(* CODESYS project shutter.library
   Company: ESO
   Description: Local Device Control - LDC Shutter Library based on State Machine
   Version: 1.1.1.0
   Placeholder: ESO LDC Shutter Library
   Author: Dan Popovic
   Title: ESO LDC Shutter Library

Project tree, tasks and I/O mapping:
  libraries: Tc2_Standard, * (Beckhoff Automation GmbH); Tc2_System, * (Beckhoff Automation GmbH); Tc3_EventLogger, * (Beckhoff Automation GmbH); Tc3_Module, * (Beckhoff Automation GmbH); VisuDialogs, * (System); VisuSymbols, 3.5.10.0 (System)
  config/
    Device1_EtherCAT_SPLC014.xti
    Mappings_HW_SPLC014.xml
    Mappings_SIM.xml
  00000000-0000-0000-0000-000000000000|config\Device1_EtherCAT_SPLC014.xti
  00000000-0000-0000-0000-000000000000|config\Mappings_HW_SPLC014.xml
  00000000-0000-0000-0000-000000000000|config\Mappings_SIM.xml
  doc/
  DUTs/
    Enumerated/
      data type E_SHUTTER_COMMAND
      data type E_SHUTTER_ERROR
      data type E_SHUTTER_EVENT
      data type E_SHUTTER_HW_STATUS
      data type E_SHUTTER_RPC_ERROR
      data type E_SHUTTER_STATE
      data type E_SHUTTER_STATUS
      data type E_SHUTTER_SUBSTATE
    Structures/
      data type T_SHUTTER_CFG
      data type T_SHUTTER_CTRL
      data type T_SHUTTER_INFO
      data type T_SHUTTER_STAT
      data type T_SIM_SHUTTER_CFG
      data type T_SIM_SHUTTER_STAT
  GVLs/
  lib/
  POUs/
    function block FB_SHUTTER [ST]: ActionCloseExecute, ActionDisableComplete, ActionDisableExecute, ActionEnableComplete, ActionErrExecute, ActionInitAbort, ActionInitComplete, ActionInitExecute, ActionInitReject, ActionOpenExecute, ActionResetExecute, ActionStopExecute, ActionUnexpExecute, ActivityClosing, ActivityDisabling, ActivityInitializing, ActivityOpening, CheckForEvents, M_GetLogicalState, M_GetRpcErrorText, M_SetLastCommand, M_SetRpcStatus, RPC_Close, RPC_Disable, RPC_Enable, RPC_Init, RPC_Open, RPC_Reset, RPC_SetDebug, RPC_SetLog, RPC_Stop
    function block FB_SHUTTER_BASE [ST]: ActionCloseExecute, ActionDisableExecute, ActionEnableComplete, ActionEnableExecute, ActionErrExecute, ActionInitAbort, ActionInitComplete, ActionInitExecute, ActionInitReject, ActionOpenExecute, ActionResetExecute, ActionStopExecute, ActionUnexpExecute, ActivityClosing, ActivityDisabling, ActivityInitializing, ActivityOpening, CheckForEvents, M_Configure, M_GetErrorText, M_LogEventDebug, M_LogEventEnd, M_LogEventError, M_LogEventGeneral, M_LogEventStart, M_SetStatus, ProcessEvents, SetAction, SetEvent, SetState
    function block FB_SIM_SHUTTER [ST]: M_GetLogicalState, RPC_ResetConfig, RPC_SetActiveLow_Closed, RPC_SetActiveLow_Fault, RPC_SetActiveLow_Open, RPC_SetActiveLow_Switch, RPC_SetCouplerState, RPC_SetDelay, RPC_SetFault, SetState
    program MAIN [ST]
  Version/
    global variables Global_Version
  VISUs/
    Templates/
      visualisation GUI_TEMPLATE_SHUTTER
    visualisation GUI_All
    visualisation GUI_Shutter001
  text list GlobalTextList
  00000000-0000-0000-0000-000000000000|Shutter.tmc
  Shutter.tmc
*)

// DUTs/Enumerated/E_SHUTTER_COMMAND
{attribute 'qualified_only'}
{attribute 'strict'}
TYPE E_SHUTTER_COMMAND :
(
	NONE	:= 0,
	
	RESET,
	INIT,
	STOP,
	ENABLE,
	DISABLE,
	OPEN,
	CLOSE
	
);
END_TYPE

// DUTs/Enumerated/E_SHUTTER_ERROR
{attribute 'qualified_only'}
{attribute 'strict'}
TYPE E_SHUTTER_ERROR :
(
	OK						:= 0,
	HW_NOT_OP,			
	INIT_FAILURE,		
	UNEXPECTED_CLOSED,
	UNEXPECTED_NONE,
	UNEXPECTED_OPENED,
	FAULT_SIG,
	BOTH_SIG_ACTIVE,
	TIMEOUT_ENABLE,
	TIMEOUT_DISABLE,
	TIMEOUT_INIT,
	TIMEOUT_CLOSE,
	TIMEOUT_OPEN,

	SIM_NOT_INITIALISED		:= 90,
	SIM_NULL_POINTER			:= 100	// Simulator error
);
END_TYPE

// DUTs/Enumerated/E_SHUTTER_EVENT
{attribute 'qualified_only'}
{attribute 'strict'}
TYPE E_SHUTTER_EVENT :
(
	NONE	:= 0,
	
	(* events corresponding to commands *)
	RESET,
	INIT,
	STOP,
	ENABLE,
	DISABLE,
	OPEN,
	CLOSE,
	
	(* 
		Events corresponding to internal events 
	*)
	
	INITOPEN,		// Needed for detection of HW failures during initialisation
	INITCLOSED,
	DISABLEOPEN,
	DISABLECLOSED,
	
	(* events mapped to HW signals *)
	ISOPEN,
	ISCLOSED,

	HWOK,
	ERRHW,
	ERRFAULT,
	ERRALLACTIVE,
	ERRNONEACTIVE,	
	ERRINIT,
	ERRDISABLE,
	ERRTIMEOUTCLOSE,
	ERRTIMEOUTOPEN
	
);
END_TYPE

// DUTs/Enumerated/E_SHUTTER_HW_STATUS
{attribute 'qualified_only'}
{attribute 'strict'}
TYPE E_SHUTTER_HW_STATUS :
(
	UNKNOWN	:= 0,
	ERROR,
	CLOSED,
	OPEN
);
END_TYPE

// DUTs/Enumerated/E_SHUTTER_RPC_ERROR
{attribute 'qualified_only'}
{attribute 'strict'}
TYPE E_SHUTTER_RPC_ERROR :
(
	OK					:= 0,
	NOT_OP				:= -1,			
	NOT_NOTOP_READY		:= -2,			
	NOT_NOTOP_NOTREADY	:= -3,			
	STILL_OPENING		:= -4,			
	STILL_CLOSING		:= -5,			
	LOCAL				:= -6			
);
END_TYPE

// DUTs/Enumerated/E_SHUTTER_STATE
{attribute 'qualified_only'}
{attribute 'strict'}
TYPE E_SHUTTER_STATE :
(
	NONE	:= 0,
	NOTOP,
	OP
);
END_TYPE

// DUTs/Enumerated/E_SHUTTER_STATUS
{attribute 'qualified_only'}
{attribute 'strict'}
TYPE E_SHUTTER_STATUS :
(
	OK	:= 0,
	ERROR
);
END_TYPE

// DUTs/Enumerated/E_SHUTTER_SUBSTATE
{attribute 'qualified_only'}
{attribute 'strict'}
TYPE E_SHUTTER_SUBSTATE :
(
	NONE                 	:= 0,
	
	NOTOP_NOTREADY     		:= 100,
	NOTOP_INITIALIZING		:= 102,
	NOTOP_READY_CLOSED		:= 105,
	NOTOP_READY_OPEN		:= 106,
	NOTOP_ERROR				:= 199,
	
	OP_DISABLING         	:= 205,
	OP_CLOSED				:= 212,            
	OP_CLOSING				:= 213,           
	OP_OPEN					:= 214,
	OP_OPENING				:= 215,
	OP_ERROR				:= 299
);
END_TYPE

// DUTs/Structures/T_SHUTTER_CFG
TYPE T_SHUTTER_CFG :
STRUCT
	sName:				STRING	:= 'Shutter';	// Instance name

	bActiveLowClosed:	BOOL 	:= FALSE;		// If TRUE, the CLOSED signal is Active Low, default FALSE
	bActiveLowFault:	BOOL 	:= FALSE;		// If TRUE, the FAULT signal is Active Low, default FALSE
	bActiveLowOpen:		BOOL 	:= FALSE;		// If TRUE, the OPEN signal is Active Low, default FALSE
	bActiveLowSwitch:	BOOL 	:= FALSE;		// If TRUE, the SWITCH signal is Active Low, default FALSE

	bIgnoreClosed:		BOOL 	:= FALSE;		// If TRUE, the CLOSED signal is Ignored, default FALSE
	bIgnoreFault:		BOOL 	:= FALSE;		// If TRUE, the FAULT signal is Ignored, default FALSE
	bIgnoreOpen:		BOOL 	:= FALSE;		// If TRUE, the OPEN signal is Ignored, default FALSE

	bInitialState:		BOOL 	:= FALSE;		// Default shutter position is FALSE/CLOSED
	nTimeout:     		UDINT 	:= 3000;		// Timeout for OPEN/CLOSE transitions [msec], default 3000 ms
	
	// Logging
	bLogExtTime:		BOOL 	:= FALSE;		// If TRUE, use external time in event logs. Default FALSE.
	bDebug:				BOOL 	:= FALSE;		// If TRUE, show event logs of Debug type. Default FALSE.
	bLog:				BOOL 	:= TRUE;		// If TRUE, log events. Default TRUE.
	
END_STRUCT
END_TYPE

// DUTs/Structures/T_SHUTTER_CTRL
TYPE T_SHUTTER_CTRL :
STRUCT
	nCommand:	E_SHUTTER_COMMAND	:= E_SHUTTER_COMMAND.NONE; (* See E_SHUTTER_COMMAND *)
	bExecute:	BOOL;
	
END_STRUCT
END_TYPE

// DUTs/Structures/T_SHUTTER_INFO
TYPE T_SHUTTER_INFO :
STRUCT
(*
Driver Information 

Change Log:
	0.1	2015-12-11	- First version - dummy implementation.
	0.2	2015-12-15	- Added timer for dummy initialization. Cleanup.
	0.3	2015-12-15	- One method per state.
	0.4	2016-06-24	- Transfer of code from FB_SHUTTER (VLT code).
	0.6 2016-06-30	- OPC UA Read Only for info and stat.
					- New method: GetLogicalState() to replace F_GET_LOGICAL_STATE
					  coming from TC3 Common.library.
					- Removed Common.library from References.
					- Implemented simulator FB_SIM_SHUTTER.
					- References are 'Always Newest'.
					- Removed Recording project.
	0.7 2016-07-01	- Added RPC_SetCouplerState() in FB_SIM_SHUTTER.
					- OPC UA Configuration cleanup
					- Removed FB_SHUTTER_SIM.
	0.8 2016-07-01	- Renaming from *_SHUTTER_* to *_SHUTTER_*.
					- Restructuring of GUI.
					- Addition of GUI Template.
					- Addition of sName as FB_SHUTTER input parameter.
					- Addition of Shutter.library
	0.9 2016-07-12	- Addition of method ActionResetExecute().
					- Errors updated only if it is currently equal to OK.
	0.10 2016-07-13	- bOpen and bClosed determined taking into account configuration.
	0.11 2017-01-25	- Addition of stat.sLastCommand.
					- Adopted Simulator from VLT FB_SIM_SHUTTER.
	0.12 2017-08-07	- Addition of BOOL return value for all RPC Calls.
					- Addition of stat.sRPCErrorText variable.
	0.13 2017-08-25	- Improved RPC Calls for all possible failures.
	0.14 2017-08-25	- Removed E_SHUTTER_SUBSTATE.NOTOP_READY substate.
					- Fixed RPC_Enable bug.
	0.15.0.0		- Single pointer to simulator
					- Updated Visualisation version
	0.16.0.0		- Corrected Simulator handling of Update.
					- Removed bUpdate variable from Simulator.
					- Addition of SetState() Simulator method.
	0.17.0.0		- Simulator delay set to half real shutter timeout.
	0.18.0.0		- Addition of all cfg params as input params.
					- Addition of M_Configure() in FB_SHUTTER_BASE.
					- Added return value for Simulator RPC calls.
					- Added small delay to simulator on re-boot.
					- Moved sName to cfg structure.
					- Single GUI for all shutters.
	0.19.0.0		- Addition of measured times for open/close in T_SHUTTER_STAT.
	0.20.0.0		- Addition of stat.sLibVersion
	0.21.0.0		- RPC calls return INT.
					- Addition of E_SHUTTER_RPC_ERROR.
	0.22.0.0		- Addition of M_GetRpcErrorText().
					- Addition of M_SetRpcStatus().
					- Improved template GUI.
					- Addition of M_GetErrorText().
					- M_SetStatus() replaced SetStatus().
					- Improved error handling.
	0.22.0.1		- Addition of library category ESO/ELT.
	0.23.0.0		- Renaming States STANDBY->NOTOP & FAILURE->ERROR.
					- RPC commands rejected in Local mode.
	0.23.0.1		- Corrected handling of IgnoreFault.
	1.0.0.0			- WARNING: Requires TwinCAT 3.1 build 4022.20 or higher.
					- Projects need Tc3_EventLogger library included in References.
					- Addition of Methods for Event Logs.
					- Addition of method RPC_Debug().
	1.0.0.1			- Addition of cfg.bLog flag for enable/disable of logging.
					- Renamed RPC_Debug() to RPC_SetDebug().
					- Addition of RPC_SetLog().
	1.0.0.2			- Compiled wit TwinCAT 3.1 build 4022.27.
					- Renamed TC_EVENTS.OpsEventClass to TC_EVENTS.ShutterOpsEventClass.
					- Solved problem of 'growing' libraries by setting Property/Advanced/BuildAction to None for Shutter.library.
					- Pinned ST_ShutterOpsEventClass under External Types.
	1.1.0.0			- Using Strict enumerations.
*)
	sDate:			STRING(32)	:= '2019-04-25';
	sDescription:	STRING(80) 	:= 'State Machine based Shutter controller';
	sName:			STRING(64)	:= 'FB_SHUTTER';
	sPlatform:		STRING(32)	:= 'CoDeSys';
	sSynopsis:		STRING(64)	:= 'State Machine based Shutter controller';
	nVersionMajor:	DINT		:= 1;
	nVersionMinor:	DINT		:= 1;
END_STRUCT
END_TYPE

// DUTs/Structures/T_SHUTTER_STAT
TYPE T_SHUTTER_STAT :
STRUCT
	//
	// Common variables START
	//
	bLocal:			BOOL	:= FALSE;						(* Device operated from PLC GUI *)

	nState:			E_SHUTTER_STATE		:= E_SHUTTER_STATE.NOTOP;			(* State, see E_SHUTTER_STATE *)
	nSubstate:		E_SHUTTER_SUBSTATE	:= E_SHUTTER_SUBSTATE.NOTOP_NOTREADY;(* Substate, see E_SHUTTER_SUBSTATE *)

	nErrorCode: 	E_SHUTTER_ERROR 	:= E_SHUTTER_ERROR.OK;				(* Error code *)
	nLastCommand:	E_SHUTTER_COMMAND	:= E_SHUTTER_COMMAND.NONE;			(* Last command sent to the device *)
	nStatus: 		E_SHUTTER_STATUS	:= E_SHUTTER_STATUS.OK; 			(* Device status *)
	nHwStatus: 		E_SHUTTER_HW_STATUS	:= E_SHUTTER_HW_STATUS.UNKNOWN; 	(* Unknown, error, open, closed. See E_SHUTTER_HW_STATUS *)
	nRpcErrorCode: 	E_SHUTTER_RPC_ERROR := E_SHUTTER_RPC_ERROR.OK;			(* RPC Error code *)

	sState:			STRING	:= 'NOT OP';					(* State textual description *)
	sSubstate:		STRING	:= 'NOT READY';					(* Substate textual description *)
	sErrorText: 	STRING 	:= 'OK'; 						(* Error text *)
	sRPCErrorText: 	STRING 	:= 'OK'; 						(* RPC Error text *)
	sStatus: 		STRING 	:= 'OK'; 						(* Status in textual form, e.g. 'OFF' *)
	sHwStatus: 		STRING 	:= 'UNKNOWN'; 					(* HW Status in textual form: 'UNKNOWN', 'ERROR', 'OPEN' or 'CLOSED' *)
	sLastCommand:	STRING	:= 'NONE';						(* Last command, as string, sent to the device *)
	sLibVersion:	STRING	:= 'UNKNOWN';					(* Library version as string, e.g. '1.2.0.0' *)
	
	sActionDesc:	STRING	:= '';
	sEventDesc:		STRING	:= '';

	nCycleCounter:	UDINT	:= 0;							// Alive flag
	nCycleTime:		UDINT	:= 0;							// Cycle time in us (microsec)
	//
	// Common variables END
	//

	//
	// Device specific variables
	//
	nLastTimeToOpen:	DINT	:= -1;	// Time taken for last OPEN command [msec] (-1 = failure)
	nLastTimeToClose:	DINT	:= -1;	// Time taken for last CLOSE command [msec] (-1 = failure)
END_STRUCT
END_TYPE

// DUTs/Structures/T_SIM_SHUTTER_CFG
TYPE T_SIM_SHUTTER_CFG :
STRUCT
	bActiveLowClosed:	BOOL := FALSE;
	bActiveLowFault:	BOOL := FALSE;
	bActiveLowOpen:		BOOL := FALSE;
	bActiveLowSwitch:	BOOL := FALSE;

	nDelay:     		UDINT := 2000;	(* Simulated delay for commands [msec] *)
	
END_STRUCT
END_TYPE

// DUTs/Structures/T_SIM_SHUTTER_STAT
TYPE T_SIM_SHUTTER_STAT :
STRUCT
	bInitialised:	BOOL	:= FALSE;						(* If TRUE, shutter simulator is initialised *)

	nErrorCode: 	DINT 	:= E_SHUTTER_ERROR.SIM_NOT_INITIALISED;	(* Error code *)
	sErrorText: 	STRING 	:= 'NOT INITIALISED'; 			(* Error text *)
	sStatus: 		STRING 	:= 'ERROR'; 					(* Shutter status in textual form, e.g. 'OFF' *)
END_STRUCT
END_TYPE

// Version/Global_Version
{attribute 'TcGenerated'}
{attribute 'no-analysis'}
{attribute 'linkalways'}
// This function has been automatically generated from the project information.
VAR_GLOBAL CONSTANT
	{attribute 'const_non_replaced'}
	stLibVersion_ESO_LDC_Shutter_Library : ST_LibVersion := (iMajor := 1, iMinor := 1, iBuild := 1, iRevision := 0, nFlags := 0, sVersion := '1.1.1.0');
END_VAR

// POUs/FB_SHUTTER
FUNCTION_BLOCK FB_SHUTTER EXTENDS FB_SHUTTER_BASE
VAR_INPUT
END_VAR
VAR_OUTPUT
END_VAR
VAR
	
	(***** Local variables *****)
	{attribute 'OPC.UA.DA' := '0'}
	toutCmd:	TON;
	{attribute 'OPC.UA.DA' := '0'}
	bOpen:		BOOL;
	{attribute 'OPC.UA.DA' := '0'}
	bClosed:	BOOL;
	{attribute 'OPC.UA.DA' := '0'}
	bFault: 	BOOL;

	(***** Physical signals - to be mapped!!! *****)

	(* Outputs *)
	{attribute 'OPC.UA.DA' := '0'}
	q_bSwitch 		AT %Q*: 		BOOL;

	(* Inputs *)	
	{attribute 'OPC.UA.DA' := '0'}
	i_nCouplerState	AT %I*: 		UINT := 8;	(* Link it to Coupler->InfoData->State *)
	{attribute 'OPC.UA.DA' := '0'}
	i_bFault 		AT %I*: 		BOOL;
	{attribute 'OPC.UA.DA' := '0'}
	i_bOpen 		AT %I*: 		BOOL;
	{attribute 'OPC.UA.DA' := '0'}
	i_bClosed		AT %I*: 		BOOL;

END_VAR

// Execute the base class object FB_SHUTTER_BASE
SUPER^();

METHOD ActionCloseExecute
VAR_INPUT
END_VAR
(* code to initiate the closing of the shutter *)
SetAction('ActionCloseExecute');

// Log event
M_LogEventStart('CLOSE');

(* Clear the error *)
M_SetStatus(E_SHUTTER_ERROR.OK);

(* Close the shutter *)
q_bSwitch	:= M_GetLogicalState(FALSE, cfg.bActiveLowSwitch);

(* start the timer *)
toutCmd(IN:=FALSE);
toutCmd(IN:=TRUE,PT:=UDINT_TO_TIME(cfg.nTimeout));
END_METHOD

METHOD ActionDisableComplete
VAR_INPUT
END_VAR
SetAction('ActionDisableComplete');

(* reply OK *)
M_SetStatus(E_SHUTTER_ERROR.OK);

(* Reset the timer action *)
toutCmd(IN:=FALSE);
END_METHOD

METHOD ActionDisableExecute
VAR_INPUT
END_VAR
SetAction('ActionDisableExecute');

// Log event
M_LogEventStart('DISABLE');

(* Set Shutter initial position obtained from the configuration *)
q_bSwitch	:= M_GetLogicalState(cfg.bInitialState, cfg.bActiveLowSwitch);

(* start the cmd timer *)
toutCmd(IN:=FALSE);
toutCmd(IN:=TRUE,PT:=UDINT_TO_TIME(cfg.nTimeout));
END_METHOD

METHOD ActionEnableComplete
VAR_INPUT
END_VAR
SetAction('ActionEnableComplete');

// Log event
M_LogEventEnd('ENABLE');

(* reply OK *)
M_SetStatus(E_SHUTTER_ERROR.OK);

(* Reset the timer action *)
toutCmd(IN:=FALSE);
END_METHOD

METHOD ActionErrExecute
VAR_INPUT
	nEventId:			DINT;
END_VAR
SetAction('ActionErrExecute');

IF nEvent = E_SHUTTER_EVENT.ERRFAULT THEN
	M_SetStatus(E_SHUTTER_ERROR.FAULT_SIG);	
ELSIF nEvent = E_SHUTTER_EVENT.ERRALLACTIVE THEN
	M_SetStatus(E_SHUTTER_ERROR.BOTH_SIG_ACTIVE);	
END_IF
END_METHOD

METHOD ActionInitAbort
VAR_INPUT
END_VAR
SetAction('ActionInitAbort');

(* reply Error *)
M_SetStatus(E_SHUTTER_ERROR.INIT_FAILURE);

(* Reset the timer for the command *)
toutCmd(IN:=FALSE);
END_METHOD

METHOD ActionInitComplete
VAR_INPUT
END_VAR
SetAction('ActionInitComplete');

// Log event
M_LogEventEnd('INIT');

(* reply OK *)
M_SetStatus(E_SHUTTER_ERROR.OK);

(* Reset the timer action *)
toutCmd(IN:=FALSE);
END_METHOD

METHOD ActionInitExecute
VAR_INPUT
END_VAR
SetAction('ActionInitExecute');

// Log event
M_LogEventStart('INIT');

(* Set Shutter initial position obtained from the configuration *)
q_bSwitch	:= M_GetLogicalState(cfg.bInitialState, cfg.bActiveLowSwitch);

(* start the cmd timer *)
toutCmd(IN:=FALSE);
toutCmd(IN:=TRUE,PT:=UDINT_TO_TIME(cfg.nTimeout));
END_METHOD

METHOD ActionInitReject
VAR_INPUT
END_VAR
SetAction('ActionInitReject');

(* Reject an INIT command since another one is in progress. *)
(* do not reset the timer ... *)
END_METHOD

METHOD ActionOpenExecute
VAR_INPUT
END_VAR
(* code to initiate the opening of the shutter *)

SetAction('ActionOpenExecute');

// Log event
M_LogEventStart('OPEN');

(* Clear the error *)
M_SetStatus(E_SHUTTER_ERROR.OK);

(* Open the shutter *)
q_bSwitch	:= M_GetLogicalState(TRUE, cfg.bActiveLowSwitch);

(* start the timer *)
toutCmd(IN:=FALSE);
toutCmd(IN:=TRUE,PT:=UDINT_TO_TIME(cfg.nTimeout));
END_METHOD

METHOD ActionResetExecute
VAR_INPUT
END_VAR
SetAction('ActionResetExecute');

// Log event
M_LogEventEnd('RESET');

(* reply Error *)
M_SetStatus(E_SHUTTER_ERROR.OK);

(* Disable outputs *)
q_bSwitch			:= FALSE;

(* Reset the timer for the command *)
toutCmd(IN:=FALSE);
END_METHOD

METHOD ActionStopExecute
VAR_INPUT
END_VAR
(* code to initiate the closing of the shutter *)
SetAction('ActionStopExecute');

(* Clear the error *)
M_SetStatus(E_SHUTTER_ERROR.OK);

IF stat.nSubstate = E_SHUTTER_SUBSTATE.OP_OPENING THEN
	(* Close the shutter *)
	q_bSwitch	:= M_GetLogicalState(FALSE, cfg.bActiveLowSwitch);

	// Log event
	M_LogEventEnd('STOP_CLOSE');
ELSIF stat.nSubstate = E_SHUTTER_SUBSTATE.OP_CLOSING THEN
	(* Open the shutter *)
	q_bSwitch	:= M_GetLogicalState(TRUE, cfg.bActiveLowSwitch);

	// Log event
	M_LogEventEnd('STOP_OPEN');
END_IF

(* start the timer *)
toutCmd(IN:=FALSE);
toutCmd(IN:=TRUE,PT:=UDINT_TO_TIME(cfg.nTimeout));
END_METHOD

METHOD ActionUnexpExecute
VAR_INPUT
	nEventId:			DINT;
END_VAR
SetAction('ActionUnexpExecute');

(*
	We don't want to overwrite initial error.
	Update error only if it is currently equal to OK. 
*)
IF stat.nErrorCode = E_SHUTTER_ERROR.OK THEN
	IF nEvent = E_SHUTTER_EVENT.ISOPEN THEN
		M_LogEventError('Shutter unexpectedly OPEN');
		M_SetStatus(E_SHUTTER_ERROR.UNEXPECTED_OPENED);
	ELSIF nEvent = E_SHUTTER_EVENT.ISCLOSED THEN
		M_LogEventError('Shutter unexpectedly CLOSED');
		M_SetStatus(E_SHUTTER_ERROR.UNEXPECTED_CLOSED);
	ELSIF nEvent = E_SHUTTER_EVENT.ERRNONEACTIVE THEN
		M_LogEventError('Both Shutter end switches unexpectedly cleared');
		M_SetStatus(E_SHUTTER_ERROR.UNEXPECTED_NONE);
	END_IF
END_IF
END_METHOD

METHOD ActivityClosing
VAR_INPUT
END_VAR
(* 
	This activity monitors the close shutter task and 
	triggers the ISOPEN event at completion. 
*)
SetAction('ActivityClosing');

(* 
	if the timeout is detected before reaching the position, 
	then trigger the internal error event 
*)
toutCmd(IN:=TRUE);
IF toutCmd.Q THEN
	// Log event
	M_LogEventError('CLOSE command timed out');

	// Set the time to CLOSE to -1, meaning FAILED
	stat.nLastTimeToClose	:= -1;
	
	toutCmd(IN:=FALSE);	(* Reset Timer *)
	nInternalEvent  := E_SHUTTER_EVENT.ERRTIMEOUTCLOSE;
	M_SetStatus(E_SHUTTER_ERROR.TIMEOUT_CLOSE);
END_IF

// Check if shutter is CLOSED
IF 	((bOpen   = FALSE OR  cfg.bIgnoreOpen) AND bClosed = TRUE)  OR
	( bOpen   = FALSE AND cfg.bIgnoreClosed) THEN
	// Log event
	M_LogEventEnd('CLOSE');

	// Get the time to CLOSE
	// The actual time equals the measured time minus a PLC task cycle.
	stat.nLastTimeToClose := TIME_TO_DINT(toutCmd.ET) - UDINT_TO_DINT(stat.nCycleTime)/1000;
	
	toutCmd(IN:=FALSE);	// Reset Timer
	nEvent 	:= E_SHUTTER_EVENT.ISCLOSED;
	M_SetStatus(E_SHUTTER_ERROR.OK);	
	RETURN;
END_IF
END_METHOD

METHOD ActivityDisabling
VAR_INPUT
END_VAR
(* 
	Activity to monitor the shutter disabling task. 
	The end state should be the predefined position of the shutter
	that is defined by configuration parameter cfg.bInitialState.
*)
SetAction('ActivityDisabling');

(* check if the initial position is reached *)
IF cfg.bInitialState = FALSE THEN
	(* Waiting for CLOSED state *)
	IF	(bOpen   = FALSE AND (bClosed = TRUE OR cfg.bIgnoreClosed))		OR
		(bClosed = TRUE  AND cfg.bIgnoreOpen) 	THEN
		// Log event
		M_LogEventDebug('After DISABLE the shutter should be CLOSED');
		M_LogEventEnd('DISABLE_CLOSE');

		nEvent  := E_SHUTTER_EVENT.DISABLECLOSED;
		M_SetStatus(E_SHUTTER_ERROR.OK);
		RETURN;
	END_IF
ELSE
	(* Waiting for OPEN state *)
	IF	(bOpen   = TRUE  AND (bClosed = FALSE OR cfg.bIgnoreClosed))	OR
		(bClosed = FALSE AND cfg.bIgnoreOpen) 	THEN
		// Log event
		M_LogEventDebug('After DISABLE the shutter should be OPEN');
		M_LogEventEnd('DISABLE_OPEN');

		nEvent  := E_SHUTTER_EVENT.DISABLEOPEN;
		M_SetStatus(E_SHUTTER_ERROR.OK);
		RETURN;
	END_IF		
END_IF


(* 
	if the timeout is detected before reaching the target position, 
	then trigger the internal error event 
*)
toutCmd(IN:=TRUE);
IF toutCmd.Q THEN
	// Log event
	M_LogEventError('DISABLE command timed out');

	toutCmd(IN:=FALSE);	(* Reset the timer *)
	nEvent  := E_SHUTTER_EVENT.ERRDISABLE;
	M_SetStatus(E_SHUTTER_ERROR.TIMEOUT_DISABLE);
END_IF
END_METHOD

METHOD ActivityInitializing
VAR_INPUT
END_VAR
(* 
	Activity to monitor the shutter initialization task and 
	trigger the E_SHUTTER_EVENT.INITCLOSED or E_SHUTTER_EVENT.INITOPEN event depending 
	on the configured default state. 		
*)
SetAction('ActivityInitializing');


(* 
	Check if the initial position is reached.
	We need additional internal events E_SHUTTER_EVENT.INITCLOSED & E_SHUTTER_EVENT.INITOPEN in order to
	cope with the scenario when the initial state is the oposit one from the configured target.
	Example:
		The shutter ISCLOSED at the beginning of this activity while the configured default state ISCLOSED.
		By introducing E_SHUTTER_EVENT.INITCLOSED & E_SHUTTER_EVENT.INITOPEN we avoid the ISCLOSED event.
*)
IF cfg.bInitialState = FALSE THEN
	(* Waiting for CLOSED state *)
	IF	(bOpen   = FALSE AND (bClosed = TRUE OR cfg.bIgnoreClosed))		OR
		(bClosed = TRUE  AND cfg.bIgnoreOpen) 	THEN
		nInternalEvent  := E_SHUTTER_EVENT.INITCLOSED;
	END_IF
ELSE
	(* Waiting for OPEN state *)
	IF	(bOpen   = TRUE  AND (bClosed = FALSE OR cfg.bIgnoreClosed))	OR
		(bClosed = FALSE AND cfg.bIgnoreOpen) 	THEN
		nInternalEvent  := E_SHUTTER_EVENT.INITOPEN;
	END_IF		
END_IF


(* 
	If the timeout is detected before reaching the initial position, 
	then trigger the internal error event 
*)
toutCmd(IN:=TRUE);
IF toutCmd.Q THEN
	// Log event
	M_LogEventError('INIT command timed out');

	toutCmd(IN:=FALSE);	(* Reset the timer *)
	nInternalEvent  := E_SHUTTER_EVENT.ERRINIT;
	M_SetStatus(E_SHUTTER_ERROR.TIMEOUT_INIT);
END_IF
END_METHOD

METHOD ActivityOpening
VAR_INPUT
END_VAR
(* 
	This activity to monitor the open shutter task and 
	trigger the ISOPEN event at completion. 
*)
SetAction('ActivityOpening');

(* 
	if the timeout is detected before reaching the position, 
	then trigger the internal error event 
*)
toutCmd(IN:=TRUE);
IF toutCmd.Q THEN
	// Log event
	M_LogEventError('OPEN command timed out');

	// Set the time to OPEN to -1, meaning FAILED
	stat.nLastTimeToOpen	:= -1;
	
	toutCmd(IN:=FALSE);	(* Reset Timer *)
	nInternalEvent  := E_SHUTTER_EVENT.ERRTIMEOUTOPEN;
	M_SetStatus(E_SHUTTER_ERROR.TIMEOUT_OPEN);
END_IF

// Check if shutter is OPEN
IF	bOpen  THEN
	// Log event
	M_LogEventEnd('OPEN');

	// Get the time to OPEN
	// The actual time equals the measured time minus a PLC task cycle.
	stat.nLastTimeToOpen := TIME_TO_DINT(toutCmd.ET) - UDINT_TO_DINT(stat.nCycleTime)/1000;
	
	toutCmd(IN:=FALSE);	// Reset Timer
	nEvent 	:= E_SHUTTER_EVENT.ISOPEN;
	M_SetStatus(E_SHUTTER_ERROR.OK);	
	RETURN;
END_IF
END_METHOD

METHOD CheckForEvents
VAR_INPUT
END_VAR

(* 
	Start assuming the HW is OK. 
	This is needed to recover from the situation where 
	the HW was failing and now it is working.
*)
nEvent := E_SHUTTER_EVENT.HWOK;


(*
	Read all inputs, i.e. get status of INPUT signals based on ActiveLow configuration 
*)

bFault	:= M_GetLogicalState(i_bFault, 	cfg.bActiveLowFault) AND NOT cfg.bIgnoreFault;

// Get bOpen
IF 	(M_GetLogicalState(i_bOpen,   cfg.bActiveLowOpen)   = TRUE  AND NOT cfg.bIgnoreOpen) OR
	(M_GetLogicalState(i_bClosed, cfg.bActiveLowClosed) = FALSE AND NOT cfg.bIgnoreClosed AND cfg.bIgnoreOpen) THEN
	bOpen	:= TRUE;
ELSE
	bOpen	:= FALSE;
END_IF

// Get bClosed
IF 	(M_GetLogicalState(i_bOpen,   cfg.bActiveLowOpen)   = FALSE AND NOT cfg.bIgnoreOpen   AND cfg.bIgnoreClosed) OR
	(M_GetLogicalState(i_bClosed, cfg.bActiveLowClosed) = TRUE  AND NOT cfg.bIgnoreClosed) THEN
	bClosed	:= TRUE;
ELSE
	bClosed	:= FALSE;
END_IF


// HW Status in textual form: 'UNKNOWN', 'ERROR', 'OPEN' or 'CLOSED'.
// HW Status doesn't depend on the Fault signal. It's a reflection of HW Status only.
// NOTE: We don't check the error in the first 20ms of opening or closing.
IF	bOpen   = TRUE AND 
	bClosed = TRUE AND 
	(TIME_TO_UDINT(toutCmd.ET) > 20  OR TIME_TO_UDINT(toutCmd.ET) = 0)	THEN
	// Both signals active ==> ERROR
	stat.nHwStatus	:= E_SHUTTER_HW_STATUS.ERROR;
	stat.sHwStatus	:= 'ERROR';
ELSIF bOpen = FALSE AND bClosed = FALSE	THEN
	// Both signals not active ==> UNKNOWN
	stat.nHwStatus	:= E_SHUTTER_HW_STATUS.UNKNOWN;
	stat.sHwStatus	:= 'UNKNOWN';
ELSIF bOpen = TRUE  AND bClosed = FALSE	THEN
	stat.nHwStatus	:= E_SHUTTER_HW_STATUS.OPEN;
	stat.sHwStatus	:= 'OPEN';
ELSIF bOpen = FALSE AND bClosed = TRUE THEN
	stat.nHwStatus	:= E_SHUTTER_HW_STATUS.CLOSED;
	stat.sHwStatus	:= 'CLOSED';
END_IF



(* 
	Check for events in the following order: 
   	1) HW failure: without HW avilability there is no point to do anything
	2) Internal events: to allow completing the initiated commands before 
                        starting processing new commands. 
   	3) Commands: to react to external commands. Commands should be executed 
                 before processing HW signals to allow to start a recovery action.
   	4) HW signals:  such as shutter is open/closed.
*)

IF i_nCouplerState <> 8 THEN	
	(* Check if the HW is NOT OK *)
	(*
	If the hardware status is NOT OK, we cannot trust the readings.
	Variable i_nCouplerState has to be mapped to a State of a terminal, e.g. EK1100.
	The value should be 8.
	NOTE: We don't check in first 500 cycles so EtherCAT gets stable.
 	*)
	SetEvent(E_SHUTTER_EVENT.ERRHW);
	M_SetStatus(E_SHUTTER_ERROR.HW_NOT_OP);

ELSIF nInternalEvent <> E_SHUTTER_EVENT.NONE THEN
	(* Handle internal events *)
	SetEvent(nInternalEvent);
	nInternalEvent := E_SHUTTER_EVENT.NONE;
ELSIF ctrl.bExecute = TRUE  THEN
	(* Handle commands *)
	ctrl.bExecute		:= FALSE;			(* Clear the Execute bit *)
	M_SetLastCommand(ctrl.nCommand);			(* Save the last command *)
	SetEvent(ctrl.nCommand);
	ctrl.nCommand 		:= E_SHUTTER_COMMAND.NONE;	(* Clear the Command *)
ELSE
	(* Handle HW problems and unexpected bahaviour *)
	
	IF bFault = TRUE AND NOT cfg.bIgnoreFault THEN
		SetEvent(E_SHUTTER_EVENT.ERRFAULT);
		M_SetStatus(E_SHUTTER_ERROR.FAULT_SIG);
		RETURN;	
	ELSIF	(stat.nSubstate = E_SHUTTER_SUBSTATE.OP_OPENING) OR
			(stat.nSubstate = E_SHUTTER_SUBSTATE.OP_CLOSING) 	 THEN
		(* 
			In these transitioning states it should not be possible that
			both switches are active at the same time.
			When closing, the OPEN switch should deactivate before the CLOSED switch gets active.
			When opening, the CLOSED switch should deactivate before the OPEN switch gets active.
			// NOTE: We don't check the error in the first 20ms of opening or closing.
		 *) 
		IF 	bOpen = TRUE AND bClosed = TRUE AND TIME_TO_UDINT(toutCmd.ET) > 20 THEN
			SetEvent(E_SHUTTER_EVENT.ERRALLACTIVE);
			RETURN;
		END_IF
	ELSIF stat.nSubstate = E_SHUTTER_SUBSTATE.OP_CLOSING THEN
		(* 
			In this transitioning state it should not be possible that
			both switches are active at the same time.
			The OPEN switch should deactivate first. 
		*) 
		IF 	bOpen = TRUE AND bClosed = TRUE THEN
			SetEvent(E_SHUTTER_EVENT.ERRALLACTIVE);
			RETURN;
		END_IF
	END_IF

	IF stat.nSubstate = E_SHUTTER_SUBSTATE.NOTOP_READY_CLOSED OR 
	   stat.nSubstate = E_SHUTTER_SUBSTATE.NOTOP_READY_OPEN OR 
	   stat.nSubstate = E_SHUTTER_SUBSTATE.OP_DISABLING OR 
	   stat.nSubstate = E_SHUTTER_SUBSTATE.OP_CLOSED OR 
	   stat.nSubstate = E_SHUTTER_SUBSTATE.OP_OPEN OR 
	   stat.nSubstate = E_SHUTTER_SUBSTATE.OP_ERROR THEN
	   
		(* read shutter open/closed physical signals *)		
		IF	  stat.nHwStatus = E_SHUTTER_HW_STATUS.OPEN THEN
			SetEvent(E_SHUTTER_EVENT.ISOPEN);
		ELSIF stat.nHwStatus = E_SHUTTER_HW_STATUS.CLOSED THEN
			SetEvent(E_SHUTTER_EVENT.ISCLOSED);
		ELSIF bOpen = TRUE AND bClosed = TRUE THEN
			SetEvent(E_SHUTTER_EVENT.ERRALLACTIVE);
		ELSIF stat.nHwStatus	= E_SHUTTER_HW_STATUS.UNKNOWN 		AND
			  stat.nSubstate <> E_SHUTTER_SUBSTATE.OP_DISABLING	THEN
			SetEvent(E_SHUTTER_EVENT.ERRNONEACTIVE);	
		END_IF	
	END_IF	
END_IF
END_METHOD

METHOD M_GetLogicalState : BOOL
(*
	This method returns the state of the variable based on its 
	activeLow configuration.
	Syntax:
		bState	:= GetLogicalState (<var value>,  <activeLow cfg>);
		
	Example 1:
		var = TRUE;
		activeLow = FALSE;
		bState	:= GetLogicalState (TRUE,  FALSE); = TRUE

	Example 2:
		var = TRUE;
		activeLow = TRUE;
		bState	:= GetLogicalState (TRUE,  TRUE); = FALSE
*)
VAR_INPUT
	state:		BOOL;
	activeLow:	BOOL;
END_VAR
IF activeLow THEN
	M_GetLogicalState := NOT state;
ELSE
	M_GetLogicalState := state;
END_IF
END_METHOD

METHOD M_GetRpcErrorText : STRING
VAR_INPUT
	ErrorCode:	INT;
END_VAR
VAR
	str:	STRING;
END_VAR
CASE ErrorCode OF
	E_SHUTTER_RPC_ERROR.OK:					str	:= 'OK';
	E_SHUTTER_RPC_ERROR.NOT_OP:				str	:= 'Cannot control shutter. Not in OP state.';
	E_SHUTTER_RPC_ERROR.NOT_NOTOP_READY:		str	:= 'Call failed. Not in NOTOP_READY.';
	E_SHUTTER_RPC_ERROR.NOT_NOTOP_NOTREADY:	str	:= 'Call failed. Not in NOTOP_NOTREADY/ERROR.';
	E_SHUTTER_RPC_ERROR.STILL_OPENING:		str	:= 'Not allowed to close the shutter while opening.';
	E_SHUTTER_RPC_ERROR.STILL_CLOSING:		str	:= 'Not allowed to open the shutter while closing.';
	E_SHUTTER_RPC_ERROR.LOCAL:				str	:= 'RPC calls not allowed in Local mode.';
ELSE
	str	:= 'Unregistered RPC error.';
END_CASE

M_GetRpcErrorText	:= str;
END_METHOD

METHOD M_SetLastCommand
VAR_INPUT
	cmd:	E_SHUTTER_COMMAND;
END_VAR
stat.nLastCommand	:= cmd;

CASE cmd OF
	E_SHUTTER_COMMAND.RESET:
		stat.sLastCommand	:= 'RESET';
	E_SHUTTER_COMMAND.INIT:
		stat.sLastCommand	:= 'INIT';
	E_SHUTTER_COMMAND.STOP:
		stat.sLastCommand	:= 'STOP';
	E_SHUTTER_COMMAND.ENABLE:
		stat.sLastCommand	:= 'ENABLE';
	E_SHUTTER_COMMAND.DISABLE:
		stat.sLastCommand	:= 'DISABLE';
	E_SHUTTER_COMMAND.OPEN:
		stat.sLastCommand	:= 'OPEN';
	E_SHUTTER_COMMAND.CLOSE:
		stat.sLastCommand	:= 'CLOSE';
ELSE
		stat.sLastCommand	:= 'NONE';
END_CASE;
END_METHOD

METHOD M_SetRpcStatus : INT
VAR_INPUT
	nErrorCode:	E_SHUTTER_RPC_ERROR;
END_VAR
stat.nRpcErrorCode	:= nErrorCode;
stat.sRPCErrorText	:= M_GetRpcErrorText(nErrorCode);

M_SetRpcStatus		:= nErrorCode;
END_METHOD

{attribute 'TcRpcEnable':='1'}
METHOD RPC_Close : INT
VAR_INPUT
END_VAR
// RPC calls are not allowed in Local mode.
IF stat.bLocal THEN
	RPC_Close	:= M_SetRpcStatus(E_SHUTTER_RPC_ERROR.LOCAL);
	RETURN;
END_IF

// Close command is accepted only in OP state.
IF stat.nState <> E_SHUTTER_STATE.OP THEN
	RPC_Close	:= M_SetRpcStatus(E_SHUTTER_RPC_ERROR.NOT_OP);
	RETURN;
END_IF

// Shutter should not be commanded to close while still opening.
IF stat.nSubstate = E_SHUTTER_SUBSTATE.OP_OPENING THEN
	RPC_Close	:= M_SetRpcStatus(E_SHUTTER_RPC_ERROR.STILL_OPENING);
	RETURN;
END_IF

ctrl.nCommand := E_SHUTTER_COMMAND.CLOSE;
ctrl.bExecute := TRUE;

// Call was successful
RPC_Close	:= M_SetRpcStatus(E_SHUTTER_RPC_ERROR.OK);
END_METHOD

{attribute 'TcRpcEnable':='1'}
METHOD RPC_Disable : INT
VAR_INPUT
END_VAR
// RPC calls are not allowed in Local mode.
IF stat.bLocal THEN
	RPC_Disable	:= M_SetRpcStatus(E_SHUTTER_RPC_ERROR.LOCAL);
	RETURN;
END_IF

// Disable command is accepted only if device is in OP state.
IF stat.nState <> E_SHUTTER_STATE.OP THEN
	RPC_Disable	:= M_SetRpcStatus(E_SHUTTER_RPC_ERROR.NOT_OP);
	RETURN;
END_IF

ctrl.nCommand := E_SHUTTER_COMMAND.DISABLE;
ctrl.bExecute := TRUE;

// Call was successful
RPC_Disable	:= M_SetRpcStatus(E_SHUTTER_RPC_ERROR.OK);
END_METHOD

{attribute 'TcRpcEnable':='1'}
METHOD RPC_Enable : INT
VAR_INPUT
END_VAR
// RPC calls are not allowed in Local mode.
IF stat.bLocal THEN
	RPC_Enable	:= M_SetRpcStatus(E_SHUTTER_RPC_ERROR.LOCAL);
	RETURN;
END_IF

// Enable command is accepted only if device is in NOTOP_READY.
IF	stat.nState = E_SHUTTER_STATE.NOTOP						AND  
	stat.nSubstate <> E_SHUTTER_SUBSTATE.NOTOP_READY_OPEN	AND  
	stat.nSubstate <> E_SHUTTER_SUBSTATE.NOTOP_READY_CLOSED		THEN
	RPC_Enable	:= M_SetRpcStatus(E_SHUTTER_RPC_ERROR.NOT_NOTOP_READY);
	RETURN;
END_IF

ctrl.nCommand := E_SHUTTER_COMMAND.ENABLE;
ctrl.bExecute := TRUE;

// Call was successful
RPC_Enable	:= M_SetRpcStatus(E_SHUTTER_RPC_ERROR.OK);
END_METHOD

{attribute 'TcRpcEnable':='1'}
METHOD RPC_Init : INT
VAR_INPUT
END_VAR
// RPC calls are not allowed in Local mode.
IF stat.bLocal THEN
	RPC_Init	:= M_SetRpcStatus(E_SHUTTER_RPC_ERROR.LOCAL);
	RETURN;
END_IF

// Init command is accepted only if device is in NOTOP_NOTREADY or ERROR.
IF 	stat.nSubstate <> E_SHUTTER_SUBSTATE.NOTOP_NOTREADY  AND  
	stat.nSubstate <> E_SHUTTER_SUBSTATE.NOTOP_ERROR 		THEN
	RPC_Init	:= M_SetRpcStatus(E_SHUTTER_RPC_ERROR.NOT_NOTOP_NOTREADY);
	RETURN;
END_IF

ctrl.nCommand := E_SHUTTER_COMMAND.INIT;
ctrl.bExecute := TRUE;


// Call was successful
RPC_Init	:= M_SetRpcStatus(E_SHUTTER_RPC_ERROR.OK);
END_METHOD

{attribute 'TcRpcEnable':='1'}
METHOD RPC_Open : INT
VAR_INPUT
END_VAR
// RPC calls are not allowed in Local mode.
IF stat.bLocal THEN
	RPC_Open	:= M_SetRpcStatus(E_SHUTTER_RPC_ERROR.LOCAL);
	RETURN;
END_IF

// Open command is accepted only in OP state.
IF stat.nState <> E_SHUTTER_STATE.OP THEN
	RPC_Open	:= M_SetRpcStatus(E_SHUTTER_RPC_ERROR.NOT_OP);
	RETURN;
END_IF

// Shutter should not be commanded to open while still closing.
IF stat.nSubstate = E_SHUTTER_SUBSTATE.OP_CLOSING THEN
	RPC_Open	:= M_SetRpcStatus(E_SHUTTER_RPC_ERROR.STILL_CLOSING);
	RETURN;
END_IF

ctrl.nCommand := E_SHUTTER_COMMAND.OPEN;
ctrl.bExecute := TRUE;

// Call was successful
RPC_Open	:= M_SetRpcStatus(E_SHUTTER_RPC_ERROR.OK);
END_METHOD

{attribute 'TcRpcEnable':='1'}
METHOD RPC_Reset : INT
VAR_INPUT
END_VAR
// RPC calls are not allowed in Local mode.
IF stat.bLocal THEN
	RPC_Reset	:= M_SetRpcStatus(E_SHUTTER_RPC_ERROR.LOCAL);
	RETURN;
END_IF

ctrl.nCommand := E_SHUTTER_COMMAND.RESET;
ctrl.bExecute := TRUE;

// Call was successful
RPC_Reset	:= M_SetRpcStatus(E_SHUTTER_RPC_ERROR.OK);
END_METHOD

{attribute 'TcRpcEnable':='1'}
METHOD RPC_SetDebug : INT
VAR_INPUT
	in_bDebug:	BOOL 	:= FALSE;		// If TRUE, show event logs of Debug type
END_VAR
// Enable/disable Debugging
cfg.bDebug	:= in_bDebug;

// Call was successful
RPC_SetDebug	:= M_SetRpcStatus(E_SHUTTER_RPC_ERROR.OK);
END_METHOD

{attribute 'TcRpcEnable':='1'}
METHOD RPC_SetLog : INT
VAR_INPUT
	in_bLog:	BOOL 	:= FALSE;		// If TRUE, activate event logging
END_VAR
// Enable/disable Logging
cfg.bLog	:= in_bLog;

// Call was successful
RPC_SetLog	:= M_SetRpcStatus(E_SHUTTER_RPC_ERROR.OK);
END_METHOD

{attribute 'TcRpcEnable':='1'}
METHOD RPC_Stop : INT
VAR_INPUT
END_VAR
// RPC calls are not allowed in Local mode.
IF stat.bLocal THEN
	RPC_Stop	:= M_SetRpcStatus(E_SHUTTER_RPC_ERROR.LOCAL);
	RETURN;
END_IF

ctrl.nCommand := E_SHUTTER_COMMAND.STOP;
ctrl.bExecute := TRUE;

// Call was successful
RPC_Stop	:= M_SetRpcStatus(E_SHUTTER_RPC_ERROR.OK);
END_METHOD

END_FUNCTION_BLOCK

// POUs/FB_SHUTTER_BASE
FUNCTION_BLOCK FB_SHUTTER_BASE
VAR_INPUT
	{attribute 'OPC.UA.DA':='0'}
	in_sName:				STRING	:= 'Shutter';	// Instance name

	{attribute 'OPC.UA.DA':='0'}
	in_bActiveLowClosed:	BOOL 	:= FALSE;		// If TRUE, the CLOSED signal is Active Low, default FALSE
	{attribute 'OPC.UA.DA':='0'}
	in_bActiveLowFault:		BOOL 	:= FALSE;		// If TRUE, the FAULT signal is Active Low, default FALSE
	{attribute 'OPC.UA.DA':='0'}
	in_bActiveLowOpen:		BOOL 	:= FALSE;		// If TRUE, the OPEN signal is Active Low, default FALSE
	{attribute 'OPC.UA.DA':='0'}
	in_bActiveLowSwitch:	BOOL 	:= FALSE;		// If TRUE, the SWITCH signal is Active Low, default FALSE

	{attribute 'OPC.UA.DA':='0'}
	in_bIgnoreClosed:		BOOL 	:= FALSE;		// If TRUE, the CLOSED signal is Ignored, default FALSE
	{attribute 'OPC.UA.DA':='0'}
	in_bIgnoreFault:		BOOL 	:= FALSE;		// If TRUE, the FAULT signal is Ignored, default FALSE
	{attribute 'OPC.UA.DA':='0'}
	in_bIgnoreOpen:			BOOL 	:= FALSE;		// If TRUE, the OPEN signal is Ignored, default FALSE

	
	{attribute 'OPC.UA.DA':='0'}
	in_bInitialState:		BOOL 	:= FALSE;		// Default shutter position is FALSE/CLOSED
	{attribute 'OPC.UA.DA':='0'}
	in_nTimeout:     		UDINT 	:= 3000;		// Timeout for OPEN/CLOSE transitions [msec], default 3000 ms

	{attribute 'OPC.UA.DA':='0'}
	in_bLogExtTime:			BOOL 	:= FALSE;		// If TRUE, use external time in event logs. Default FALSE.
	{attribute 'OPC.UA.DA':='0'}
	in_bLog:				BOOL 	:= TRUE;		// If TRUE, log events. Default TRUE.
END_VAR
VAR_OUTPUT
END_VAR
VAR RETAIN
END_VAR
VAR
	{attribute 'OPC.UA.DA' := '1'}
	cfg:		T_SHUTTER_CFG;	
	{attribute 'OPC.UA.DA' := '1'}
	ctrl:		T_SHUTTER_CTRL;	
	{attribute 'OPC.UA.DA' := '1'}
	{attribute 'OPC.UA.DA.Access' := '1'}
	info:		T_SHUTTER_INFO;	(* ReadOnly *)
	{attribute 'OPC.UA.DA' := '1'}
	{attribute 'OPC.UA.DA.Access' := '1'}
	stat:		T_SHUTTER_STAT;	(* ReadOnly *)

	{attribute 'OPC.UA.DA' := '0'}
	nEvent:		      	DINT := E_SHUTTER_EVENT.NONE;
	{attribute 'OPC.UA.DA' := '0'}
	nInternalEvent:		DINT := E_SHUTTER_EVENT.NONE;
	
	// Operational Events
	{attribute 'OPC.UA.DA' := '0'}
	fbEventStart:	FB_TcMessage;
	{attribute 'OPC.UA.DA' := '0'}
	fbEventEnd:		FB_TcMessage;
	{attribute 'OPC.UA.DA' := '0'}
	fbEventError:	FB_TcMessage;
	{attribute 'OPC.UA.DA' := '0'}
	fbEventDebug:	FB_TcMessage;
	{attribute 'OPC.UA.DA' := '0'}
	fbEventGeneral:	FB_TcMessage;
	
	(***** Physical signals - to be mapped!!! *****)

	(* Outputs *)

	(* Inputs *)
	
	// Flag if the device is ready to receive commands.
	// It takes a couple of cycles for the system to read inputs after reboot.
	{attribute 'OPC.UA.DA' := '0'}
	bDeviceReady:	BOOL 	:= FALSE;

END_VAR

// On first cycle configure from input params and internally execute M_UserConfigure()
IF NOT bDeviceReady THEN
	// Set device Configuration
	M_Configure();
	RETURN;
END_IF

// Increment counter.
// This will be seen as 'alive' flag.
stat.nCycleCounter	:= stat.nCycleCounter + 1;


(* === Check for commands and internal events to be processed === *)
CheckForEvents();

(* === Process events according to the State Machine === *)
ProcessEvents();

METHOD ActionCloseExecute
VAR_INPUT
END_VAR
END_METHOD

METHOD ActionDisableExecute
VAR_INPUT
END_VAR
END_METHOD

METHOD ActionEnableComplete
VAR_INPUT
END_VAR
END_METHOD

METHOD ActionEnableExecute
VAR_INPUT
END_VAR
END_METHOD

METHOD ActionErrExecute
VAR_INPUT
	nEventId:			DINT;
END_VAR
END_METHOD

METHOD ActionInitAbort
VAR_INPUT
END_VAR
END_METHOD

METHOD ActionInitComplete
VAR_INPUT
END_VAR
END_METHOD

METHOD ActionInitExecute
VAR_INPUT
END_VAR
END_METHOD

METHOD ActionInitReject
VAR_INPUT
END_VAR
END_METHOD

METHOD ActionOpenExecute
VAR_INPUT
END_VAR
END_METHOD

METHOD ActionResetExecute
VAR_INPUT
END_VAR
END_METHOD

METHOD ActionStopExecute
VAR_INPUT
END_VAR
END_METHOD

METHOD ActionUnexpExecute
VAR_INPUT
	nEventId:			DINT;
END_VAR
END_METHOD

METHOD ActivityClosing
VAR_INPUT
END_VAR
END_METHOD

METHOD ActivityDisabling
VAR_INPUT
END_VAR
END_METHOD

METHOD ActivityInitializing
VAR_INPUT
END_VAR
END_METHOD

METHOD ActivityOpening
VAR_INPUT
END_VAR
END_METHOD

METHOD CheckForEvents
VAR_INPUT
END_VAR
END_METHOD

METHOD M_Configure : BOOL
VAR_INPUT
END_VAR
VAR
     fbGetCurTaskIdx:	GETCURTASKINDEX;
END_VAR
// If device is ready, there is nothing to configure.
IF bDeviceReady THEN
	RETURN;
END_IF

// If first cycle, copy configuration AND RETURN in order for the system to read all inputs before doing any work
IF stat.nCycleCounter = 0 THEN
	cfg.sName				:= in_sName;			// Instance name
	cfg.bActiveLowClosed	:= in_bActiveLowClosed;	// If TRUE, the CLOSED signal is Active Low, default FALSE
	cfg.bActiveLowFault		:= in_bActiveLowFault;	// If TRUE, the FAULT signal is Active Low, default FALSE
	cfg.bActiveLowOpen		:= in_bActiveLowOpen;	// If TRUE, the OPEN signal is Active Low, default FALSE
	cfg.bActiveLowSwitch	:= in_bActiveLowSwitch;	// If TRUE, the SWITCH signal is Active Low, default FALSE

	cfg.bIgnoreClosed		:= in_bIgnoreClosed;	// If TRUE, the CLOSED signal is Ignored, default FALSE
	cfg.bIgnoreFault		:= in_bIgnoreFault;		// If TRUE, the FAULT signal is Ignored, default FALSE
	cfg.bIgnoreOpen			:= in_bIgnoreOpen;		// If TRUE, the OPEN signal is Ignored, default FALSE

	cfg.bInitialState		:= in_bInitialState;	// Default shutter position is FALSE/CLOSED
	cfg.nTimeout			:= in_nTimeout;			// Timeout for OPEN/CLOSE transitions [msec], default 3000 ms

	cfg.bLogExtTime			:= in_bLogExtTime;		// If TRUE, use external time in event logs
	cfg.bLog				:= in_bLog;				// If TRUE, use external time in event logs
	
	// Get the version number 
	stat.sLibVersion	:= stLibVersion_ESO_LDC_Shutter_Library.sVersion;

	// Get cycle time in microsec.
	// CycleTime in _TaskInfo is given in 100 ns. 1 us = 1000 ns
	fbGetCurTaskIdx();
	stat.nCycleTime	:=  (TwinCAT_SystemInfoVarList._TaskInfo[fbGetCurTaskIdx.index].CycleTime)/10;
	
	// Increment counter.
	stat.nCycleCounter	:= stat.nCycleCounter + 1;
	RETURN;
ELSIF (stat.nCycleCounter * stat.nCycleTime) < 5000000 THEN
	// EtherCAT is normally ready after 3.5 sec.
	// We give it 5 sec to consider it to be ready.
	// Increment counter.
	stat.nCycleCounter	:= stat.nCycleCounter + 1;
	RETURN;
END_IF

// The system shoud be ready, i.e. coupler state is 8.

// Create Event instances
fbEventStart.CreateEx	(TC_EVENTS.ShutterOpsEventClass.ActionStart,0);
fbEventEnd.CreateEx		(TC_EVENTS.ShutterOpsEventClass.ActionEnd,0);
fbEventError.CreateEx	(TC_EVENTS.ShutterOpsEventClass.Error,0);
fbEventDebug.CreateEx	(TC_EVENTS.ShutterOpsEventClass.Debug,0);


// The device is ready now.
bDeviceReady := TRUE;


// Clear errors
M_SetStatus(E_SHUTTER_ERROR.OK);
END_METHOD

METHOD M_GetErrorText : STRING
VAR_INPUT
	ErrorCode:	DINT;
END_VAR
VAR
	str:	STRING;
END_VAR
CASE ErrorCode OF
	E_SHUTTER_ERROR.OK:					str	:= 'OK';
	E_SHUTTER_ERROR.HW_NOT_OP:			str	:= 'ERROR: TwinCAT not in OP state or CouplerState not mapped.';
	E_SHUTTER_ERROR.INIT_FAILURE:			str	:= 'ERROR: INIT command aborted due to STOP or RESET.';
	E_SHUTTER_ERROR.UNEXPECTED_CLOSED:	str	:= 'ERROR: Shutter unexpectedly closed.';
	E_SHUTTER_ERROR.UNEXPECTED_NONE:		str	:= 'ERROR: Unexpectedly no OPEN or CLOSED signal active.';
	E_SHUTTER_ERROR.UNEXPECTED_OPENED:	str	:= 'ERROR: Shutter unexpectedly opened.';
	E_SHUTTER_ERROR.FAULT_SIG:			str	:= 'ERROR: Fault signal active.';
	E_SHUTTER_ERROR.BOTH_SIG_ACTIVE:		str	:= 'ERROR: Both OPEN and CLOSED signals active.';
	E_SHUTTER_ERROR.TIMEOUT_ENABLE:		str	:= 'ERROR: ENABLE timed out.';
	E_SHUTTER_ERROR.TIMEOUT_DISABLE:		str	:= 'ERROR: DISABLE timed out.';
	E_SHUTTER_ERROR.TIMEOUT_INIT:			str	:= 'ERROR: INIT timed out.';
	E_SHUTTER_ERROR.TIMEOUT_CLOSE:		str	:= 'ERROR: CLOSE timed out.';
	E_SHUTTER_ERROR.TIMEOUT_OPEN:			str	:= 'ERROR: OPEN timed out.';
	E_SHUTTER_ERROR.SIM_NOT_INITIALISED:	str	:= 'ERROR: Shutter simulator not initialised.';
	E_SHUTTER_ERROR.SIM_NULL_POINTER:		str	:= 'ERROR: NULL pointer to Shutter.';
ELSE
	str	:= 'Unregistered error.';
END_CASE

M_GetErrorText	:= str;
END_METHOD

METHOD M_LogEventDebug : BOOL
VAR_INPUT
	sText:	STRING	:= '';
END_VAR
// Log Debug events only if both logging and debugging is enabled
IF cfg.bLog AND cfg.bDebug THEN
	fbEventDebug.ipArguments.Clear().AddString(sText);
	fbEventDebug.Send(0);
END_IF
END_METHOD

METHOD M_LogEventEnd : BOOL
VAR_INPUT
	sText:	STRING	:= '';
END_VAR
// Log only if logging is enabled
IF  NOT cfg.bLog THEN
	RETURN;
END_IF

fbEventEnd.ipArguments.Clear().AddString(sText);
fbEventEnd.Send(0);
END_METHOD

METHOD M_LogEventError : BOOL
VAR_INPUT
	sText:	STRING	:= '';
END_VAR
// Log only if logging is enabled
IF  NOT cfg.bLog THEN
	RETURN;
END_IF

fbEventError.ipArguments.Clear().AddString(sText);
fbEventError.Send(0);
END_METHOD

METHOD M_LogEventGeneral : BOOL
VAR_INPUT
	sText:	STRING	:= '';
END_VAR
// Log only if logging is enabled
IF  NOT cfg.bLog THEN
	RETURN;
END_IF

fbEventGeneral.ipArguments.Clear().AddString(sText);
fbEventGeneral.Send(0);
END_METHOD

METHOD M_LogEventStart : BOOL
VAR_INPUT
	sText:	STRING	:= '';
END_VAR
// Log only if logging is enabled
IF  NOT cfg.bLog THEN
	RETURN;
END_IF

fbEventStart.ipArguments.Clear().AddString(sText);
fbEventStart.Send(0);
END_METHOD

METHOD M_SetStatus
VAR_INPUT
	nErrorCode:	E_SHUTTER_ERROR;
END_VAR
stat.nErrorCode 	:= nErrorCode;
stat.sErrorText 	:= M_GetErrorText(nErrorCode);

IF nErrorCode <> E_SHUTTER_ERROR.OK THEN
	stat.sStatus	:= 'ERROR';
	stat.nStatus	:= E_SHUTTER_STATUS.ERROR;
ELSE
	stat.sStatus	:= 'OK';
	stat.nStatus	:= E_SHUTTER_STATUS.OK;
END_IF
END_METHOD

METHOD ProcessEvents
VAR_INPUT
END_VAR

VAR
	ActionUnexpectedOpenExecute: INT;
END_VAR

(* 
	Before processing the event, execute the Do-Activity tasks. 
	Note that, in case of orthogonal regions, more than one Do-Activity 
	could run in the same PLC cycle.
	Note: Most of these activities have timeouts since they take time.
*)

IF stat.nSubstate = E_SHUTTER_SUBSTATE.NOTOP_INITIALIZING THEN
	ActivityInitializing();
END_IF

IF stat.nSubstate = E_SHUTTER_SUBSTATE.OP_OPENING THEN
	ActivityOpening();
END_IF

IF stat.nSubstate = E_SHUTTER_SUBSTATE.OP_CLOSING THEN
	ActivityClosing();
END_IF

IF stat.nSubstate = E_SHUTTER_SUBSTATE.OP_DISABLING THEN
	ActivityDisabling();
END_IF


(* 
	Evaluate state machine transitions.
*)

CASE stat.nState OF

//***********************************
// NOTOP
//***********************************
E_SHUTTER_STATE.NOTOP:

	(* Transitions from NOTOP substates *)
	CASE stat.nSubstate OF
	
	E_SHUTTER_SUBSTATE.NOTOP_NOTREADY:		
		IF nEvent = E_SHUTTER_EVENT.INIT THEN
			ActionInitExecute();
			SetState(E_SHUTTER_STATE.NOTOP, E_SHUTTER_SUBSTATE.NOTOP_INITIALIZING);
			M_SetStatus(E_SHUTTER_ERROR.OK);
			RETURN;
		END_IF
		
	E_SHUTTER_SUBSTATE.NOTOP_INITIALIZING:			
		IF nEvent = E_SHUTTER_EVENT.STOP THEN
			ActionInitAbort();
			SetState(E_SHUTTER_STATE.NOTOP, E_SHUTTER_SUBSTATE.NOTOP_NOTREADY);
			RETURN;
		ELSIF nEvent = E_SHUTTER_EVENT.ERRINIT THEN
			SetState(E_SHUTTER_STATE.NOTOP, E_SHUTTER_SUBSTATE.NOTOP_ERROR);
			RETURN;
		ELSIF nEvent = E_SHUTTER_EVENT.INITCLOSED THEN
			ActionInitComplete();
			SetState(E_SHUTTER_STATE.NOTOP, E_SHUTTER_SUBSTATE.NOTOP_READY_CLOSED);
			RETURN;
		ELSIF nEvent = E_SHUTTER_EVENT.INITOPEN THEN
			ActionInitComplete();
			SetState(E_SHUTTER_STATE.NOTOP, E_SHUTTER_SUBSTATE.NOTOP_READY_OPEN);
			RETURN;
		END_IF
		
	E_SHUTTER_SUBSTATE.NOTOP_READY_CLOSED:			
		IF nEvent = E_SHUTTER_EVENT.ISOPEN THEN
			ActionUnexpExecute(nEvent);
			SetState(E_SHUTTER_STATE.NOTOP, E_SHUTTER_SUBSTATE.NOTOP_READY_OPEN);
			RETURN;
		ELSIF nEvent = E_SHUTTER_EVENT.ENABLE THEN
			ActionEnableComplete();
			SetState(E_SHUTTER_STATE.OP, E_SHUTTER_SUBSTATE.OP_CLOSED);
			RETURN;
		END_IF

	E_SHUTTER_SUBSTATE.NOTOP_READY_OPEN:			
		IF nEvent = E_SHUTTER_EVENT.ISCLOSED THEN
			ActionUnexpExecute(nEvent);
			SetState(E_SHUTTER_STATE.NOTOP, E_SHUTTER_SUBSTATE.NOTOP_READY_CLOSED);
			RETURN;
		ELSIF nEvent = E_SHUTTER_EVENT.ENABLE THEN
			ActionEnableComplete();
			SetState(E_SHUTTER_STATE.OP, E_SHUTTER_SUBSTATE.OP_OPEN);
			RETURN;
		END_IF

	E_SHUTTER_SUBSTATE.NOTOP_ERROR:			
		IF	nEvent = E_SHUTTER_EVENT.HWOK 				AND 
			stat.nErrorCode = E_SHUTTER_ERROR.HW_NOT_OP 	THEN
			SetState(E_SHUTTER_STATE.NOTOP, E_SHUTTER_SUBSTATE.NOTOP_NOTREADY);
			RETURN;
		END_IF
		
	END_CASE

	(* Transitions from NOTOP state *)
	IF nEvent = E_SHUTTER_EVENT.ERRHW THEN
		SetState(E_SHUTTER_STATE.NOTOP, E_SHUTTER_SUBSTATE.NOTOP_ERROR);
		RETURN;
	ELSIF nEvent = E_SHUTTER_EVENT.ERRFAULT THEN
		// TODO
		SetState(E_SHUTTER_STATE.NOTOP, E_SHUTTER_SUBSTATE.NOTOP_ERROR);			
		RETURN;
	ELSIF nEvent = E_SHUTTER_EVENT.ERRALLACTIVE THEN
		// TODO
		ActionErrExecute(nEvent);
		SetState(E_SHUTTER_STATE.NOTOP, E_SHUTTER_SUBSTATE.NOTOP_ERROR);
		RETURN;
	END_IF
	
//***********************************
// OPERATIONAL
//***********************************
E_SHUTTER_STATE.OP:

	(* Transitions from OP subastates *)
	CASE stat.nSubstate OF
	E_SHUTTER_SUBSTATE.OP_CLOSED:			
		IF nEvent = E_SHUTTER_EVENT.OPEN THEN
			ActionOpenExecute();
			SetState(E_SHUTTER_STATE.OP, E_SHUTTER_SUBSTATE.OP_OPENING);
			RETURN;
		ELSIF nEvent = E_SHUTTER_EVENT.CLOSE THEN
			// Nothing to do. Just clear previous error, if any.
			M_SetStatus(E_SHUTTER_ERROR.OK);
			RETURN;
		ELSIF nEvent = E_SHUTTER_EVENT.ISOPEN THEN
			ActionUnexpExecute(nEvent);
			SetState(E_SHUTTER_STATE.OP, E_SHUTTER_SUBSTATE.OP_OPEN);
			RETURN;
		ELSIF nEvent = E_SHUTTER_EVENT.DISABLE THEN
			ActionDisableExecute();
			SetState(E_SHUTTER_STATE.OP, E_SHUTTER_SUBSTATE.OP_DISABLING);
			RETURN;		
		ELSIF nEvent = E_SHUTTER_EVENT.ERRNONEACTIVE THEN
			ActionUnexpExecute(nEvent);
			SetState(E_SHUTTER_STATE.OP, E_SHUTTER_SUBSTATE.OP_ERROR);
			RETURN;				
		END_IF

	E_SHUTTER_SUBSTATE.OP_OPENING:			
		IF nEvent = E_SHUTTER_EVENT.ISOPEN THEN
			SetState(E_SHUTTER_STATE.OP, E_SHUTTER_SUBSTATE.OP_OPEN);
			RETURN;
		ELSIF nEvent = E_SHUTTER_EVENT.ISCLOSED THEN
			ActionUnexpExecute(nEvent);
			SetState(E_SHUTTER_STATE.OP, E_SHUTTER_SUBSTATE.OP_ERROR);
			RETURN;
		ELSIF nEvent = E_SHUTTER_EVENT.ERRTIMEOUTOPEN THEN
			SetState(E_SHUTTER_STATE.OP, E_SHUTTER_SUBSTATE.OP_ERROR);
			RETURN;
		ELSIF nEvent = E_SHUTTER_EVENT.STOP THEN
			ActionStopExecute();
			SetState(E_SHUTTER_STATE.OP, E_SHUTTER_SUBSTATE.OP_CLOSING);
			RETURN;			
		END_IF
		
	E_SHUTTER_SUBSTATE.OP_OPEN:			
		IF nEvent = E_SHUTTER_EVENT.CLOSE THEN
			ActionCloseExecute();
			SetState(E_SHUTTER_STATE.OP, E_SHUTTER_SUBSTATE.OP_CLOSING);
			RETURN;
		ELSIF nEvent = E_SHUTTER_EVENT.OPEN THEN
			// Nothing to do. Just clear previous error, if any.
			M_SetStatus(E_SHUTTER_ERROR.OK);
			RETURN;
		ELSIF nEvent = E_SHUTTER_EVENT.ISCLOSED THEN
			ActionUnexpExecute(nEvent);
			SetState(E_SHUTTER_STATE.OP, E_SHUTTER_SUBSTATE.OP_CLOSED);
			RETURN;
		ELSIF nEvent = E_SHUTTER_EVENT.DISABLE THEN
			ActionDisableExecute();
			SetState(E_SHUTTER_STATE.OP, E_SHUTTER_SUBSTATE.OP_DISABLING);
			RETURN;	
		ELSIF nEvent = E_SHUTTER_EVENT.ERRNONEACTIVE THEN
			ActionUnexpExecute(nEvent);
			SetState(E_SHUTTER_STATE.OP, E_SHUTTER_SUBSTATE.OP_ERROR);
			RETURN;				
		END_IF
		
	E_SHUTTER_SUBSTATE.OP_CLOSING:			
		IF nEvent = E_SHUTTER_EVENT.ISCLOSED THEN
			SetState(E_SHUTTER_STATE.OP, E_SHUTTER_SUBSTATE.OP_CLOSED);
			RETURN;
		ELSIF nEvent = E_SHUTTER_EVENT.ISOPEN THEN
			SetState(E_SHUTTER_STATE.OP, E_SHUTTER_SUBSTATE.OP_OPEN);
			RETURN;
		ELSIF nEvent = E_SHUTTER_EVENT.ERRTIMEOUTCLOSE THEN
			SetState(E_SHUTTER_STATE.OP, E_SHUTTER_SUBSTATE.OP_ERROR);
			RETURN;
		ELSIF nEvent = E_SHUTTER_EVENT.STOP THEN
			ActionStopExecute();
			SetState(E_SHUTTER_STATE.OP, E_SHUTTER_SUBSTATE.OP_OPENING);
			RETURN;			
		END_IF
		
	E_SHUTTER_SUBSTATE.OP_ERROR:			
		IF nEvent = E_SHUTTER_EVENT.CLOSE THEN
			ActionCloseExecute();
			SetState(E_SHUTTER_STATE.OP, E_SHUTTER_SUBSTATE.OP_CLOSING);
			RETURN;
		ELSIF nEvent = E_SHUTTER_EVENT.OPEN THEN
			ActionOpenExecute();
			SetState(E_SHUTTER_STATE.OP, E_SHUTTER_SUBSTATE.OP_OPENING);
			RETURN;			
		ELSIF nEvent = E_SHUTTER_EVENT.ISOPEN THEN
			M_LogEventGeneral('Recovered from error. Shutter is OPEN.');
			SetState(E_SHUTTER_STATE.OP, E_SHUTTER_SUBSTATE.OP_OPEN);
			RETURN;			
		ELSIF nEvent = E_SHUTTER_EVENT.ISCLOSED THEN
			M_LogEventGeneral('Recovered from error. Shutter is CLOSED.');
			SetState(E_SHUTTER_STATE.OP, E_SHUTTER_SUBSTATE.OP_CLOSED);
			RETURN;	
		ELSIF nEvent = E_SHUTTER_EVENT.DISABLE THEN
			SetState(E_SHUTTER_STATE.OP, E_SHUTTER_SUBSTATE.OP_DISABLING);
			RETURN;			
		END_IF

	E_SHUTTER_SUBSTATE.OP_DISABLING:			
		IF nEvent = E_SHUTTER_EVENT.DISABLECLOSED THEN
			SetState(E_SHUTTER_STATE.NOTOP, E_SHUTTER_SUBSTATE.NOTOP_READY_CLOSED);
			RETURN;
		ELSIF nEvent = E_SHUTTER_EVENT.DISABLEOPEN THEN
			SetState(E_SHUTTER_STATE.NOTOP, E_SHUTTER_SUBSTATE.NOTOP_READY_OPEN);
			RETURN;
		ELSIF nEvent = E_SHUTTER_EVENT.ERRDISABLE THEN
			SetState(E_SHUTTER_STATE.OP, E_SHUTTER_SUBSTATE.OP_ERROR);
			RETURN;
		END_IF
		
	END_CASE
	
	(* Transitions from OP state *)
	IF nEvent = E_SHUTTER_EVENT.ERRHW THEN
		SetState(E_SHUTTER_STATE.OP, E_SHUTTER_SUBSTATE.OP_ERROR);
		RETURN;
	ELSIF nEvent = E_SHUTTER_EVENT.ERRFAULT THEN
		SetState(E_SHUTTER_STATE.OP, E_SHUTTER_SUBSTATE.OP_ERROR);
		RETURN;
	ELSIF nEvent = E_SHUTTER_EVENT.ERRALLACTIVE THEN
		// TODO
		ActionErrExecute(nEvent);
		SetState(E_SHUTTER_STATE.OP, E_SHUTTER_SUBSTATE.OP_ERROR);
		RETURN;
	END_IF
	
END_CASE

(* 
	"Global" internal transitions valid in any state should go here.
	They do not change the active state configuration. 
	They are evaluated after all the others transitions have been 
	considered.
*) 
IF nEvent = E_SHUTTER_EVENT.RESET THEN
	ActionResetExecute();
	SetState(E_SHUTTER_STATE.NOTOP, E_SHUTTER_SUBSTATE.NOTOP_NOTREADY);
	RETURN;
END_IF
END_METHOD

METHOD SetAction
VAR_INPUT
	actionName:		STRING;
END_VAR


stat.sActionDesc := actionName;
END_METHOD

METHOD SetEvent
VAR_INPUT
	nEventId:			DINT;
END_VAR

nEvent := nEventId;

CASE nEventId OF
	E_SHUTTER_EVENT.NONE:
		stat.sEventDesc := '';
		RETURN;
		
	E_SHUTTER_EVENT.RESET:
		stat.sEventDesc := 'CMD RESET';
		RETURN;
	
	E_SHUTTER_EVENT.INIT:
		stat.sEventDesc := 'CMD INIT';
		RETURN;

	E_SHUTTER_EVENT.STOP:
		stat.sEventDesc := 'CMD STOP';
		RETURN;

	E_SHUTTER_EVENT.ENABLE:
		stat.sEventDesc := 'CMD ENABLE';
		RETURN;

	E_SHUTTER_EVENT.DISABLE:
		stat.sEventDesc := 'CMD DISABLE';
		RETURN;

	E_SHUTTER_EVENT.OPEN:
		stat.sEventDesc := 'CMD OPEN';
		RETURN;

	E_SHUTTER_EVENT.CLOSE:
		stat.sEventDesc := 'CMD CLOSE';
		RETURN;
	
	(* events corresponding to internal events *)
	E_SHUTTER_EVENT.INITCLOSED:
		stat.sEventDesc := 'INT INITCLOSED';
		RETURN;

	E_SHUTTER_EVENT.INITOPEN:
		stat.sEventDesc := 'INT INITOPEN';
		RETURN;

	E_SHUTTER_EVENT.DISABLECLOSED:
		stat.sEventDesc := 'INT DISABLECLOSED';
		RETURN;
	
	E_SHUTTER_EVENT.DISABLEOPEN:
		stat.sEventDesc := 'INT DISABLEOPEN';
		RETURN;
	
	(* evetnts mapped to HW signals *)
	E_SHUTTER_EVENT.ISOPEN:
		stat.sEventDesc := 'SIG ISOPEN';
		RETURN;

	E_SHUTTER_EVENT.ISCLOSED:
		stat.sEventDesc := 'SIG ISCLOSED';
		RETURN;

	E_SHUTTER_EVENT.HWOK:
		stat.sEventDesc := 'SIG HWOK';
		RETURN;

	E_SHUTTER_EVENT.ERRHW:
		stat.sEventDesc := 'INT ERRHW';
		RETURN;

	E_SHUTTER_EVENT.ERRFAULT:	
		stat.sEventDesc := 'INT ERRFAULT';
		RETURN;

	E_SHUTTER_EVENT.ERRALLACTIVE:
		stat.sEventDesc := 'INT ERRALLACTIVE';
		RETURN;
	
	E_SHUTTER_EVENT.ERRNONEACTIVE:	
		stat.sEventDesc := 'INT ERRNONEACTIVE';
		RETURN;
		
	E_SHUTTER_EVENT.ERRINIT:
		stat.sEventDesc := 'INT ERRINIT';
		RETURN;

	E_SHUTTER_EVENT.ERRDISABLE:
		stat.sEventDesc := 'INT ERRDISABLE';
		RETURN;
	
END_CASE 

(* INTERNAL ERROR *)
stat.sEventDesc := 'UNKNOWN EVENT';
END_METHOD

METHOD SetState : BOOL
VAR_INPUT
	nState:			E_SHUTTER_STATE;
	nSubstate:		E_SHUTTER_SUBSTATE;
END_VAR
(* 
	Update State Machine active state configuration.

	ToDo: support initial pseudo state/substate.
*)

IF nState <> E_SHUTTER_STATE.NONE THEN
	stat.nState	:= nState;
END_IF
IF nSubstate <> E_SHUTTER_SUBSTATE.NONE THEN
	stat.nSubstate	:= nSubstate;
END_IF

(* Update active state configuration description *)

IF nState = E_SHUTTER_STATE.NOTOP THEN
	stat.sState	:= 'NOT OP';
ELSIF nState = E_SHUTTER_STATE.OP THEN
	stat.sState	:= 'OPERATIONAL';
END_IF

IF nSubstate = E_SHUTTER_SUBSTATE.NOTOP_NOTREADY THEN
	stat.sSubstate	:= 'NOT READY';
ELSIF nSubstate = E_SHUTTER_SUBSTATE.NOTOP_INITIALIZING THEN
	stat.sSubstate	:= 'INITIALIAZING';
ELSIF nSubstate = E_SHUTTER_SUBSTATE.NOTOP_READY_CLOSED THEN
	stat.sSubstate	:= 'READY CLOSED';
ELSIF nSubstate = E_SHUTTER_SUBSTATE.NOTOP_READY_OPEN THEN
	stat.sSubstate	:= 'READY OPEN';
ELSIF nSubstate = E_SHUTTER_SUBSTATE.NOTOP_ERROR THEN
	stat.sSubstate	:= 'ERROR';
ELSIF nSubstate = E_SHUTTER_SUBSTATE.OP_CLOSED THEN
	stat.sSubstate	:= 'CLOSED';
ELSIF nSubstate = E_SHUTTER_SUBSTATE.OP_OPEN THEN
	stat.sSubstate	:= 'OPEN';
ELSIF nSubstate = E_SHUTTER_SUBSTATE.OP_CLOSING THEN
	stat.sSubstate	:= 'CLOSING';
ELSIF nSubstate = E_SHUTTER_SUBSTATE.OP_OPENING THEN
	stat.sSubstate	:= 'OPENING';
ELSIF nSubstate = E_SHUTTER_SUBSTATE.OP_DISABLING THEN
	stat.sSubstate	:= 'DISABLING';
ELSIF nSubstate = E_SHUTTER_SUBSTATE.OP_ERROR THEN
	stat.sSubstate	:= 'ERROR';
ELSE
	stat.sSubstate	:= '';
END_IF


SetState	:= TRUE;
END_METHOD

END_FUNCTION_BLOCK

// POUs/FB_SIM_SHUTTER
FUNCTION_BLOCK FB_SIM_SHUTTER
VAR_INPUT
	ptrDev:		POINTER TO FB_SHUTTER;
END_VAR
VAR_OUTPUT
END_VAR
VAR
	ptrCfg:		POINTER TO T_SHUTTER_CFG;
	ptrStat:	POINTER TO T_SHUTTER_STAT;

	{attribute 'OPC.UA.DA':='1'}
	cfg:			T_SIM_SHUTTER_CFG;	(* ActiveLow configuration for each signal *)
	{attribute 'OPC.UA.DA':='1'}
	stat:			T_SIM_SHUTTER_STAT;	(* Simulator status parameters *)
	
	{attribute 'OPC.UA.DA':='0'}
	bSwitch:		BOOL := FALSE;
	{attribute 'OPC.UA.DA':='0'}
	bSwitchLast:	BOOL := FALSE;
	
	{attribute 'OPC.UA.DA':='0'}
	bClosed:		BOOL := FALSE;
	{attribute 'OPC.UA.DA':='0'}
	bOpen:			BOOL := TRUE;
	{attribute 'OPC.UA.DA':='0'}
	bFault:			BOOL := FALSE;
	{attribute 'OPC.UA.DA':='0'}
	nCouplerState:	UINT := 8;       // normal coupler state
	
    (* Inputs *)
	{attribute 'OPC.UA.DA':='0'}
	i_bSwitch 		AT %I*: 		BOOL;

	(* Outputs *)	
	{attribute 'OPC.UA.DA':='0'}
	q_bFault 		AT %Q*: 		BOOL;
	{attribute 'OPC.UA.DA':='0'}
	q_bOpen 		AT %Q*: 		BOOL;
	{attribute 'OPC.UA.DA':='0'}
	q_bClosed		AT %Q*: 		BOOL;
	{attribute 'OPC.UA.DA':='0'}
	q_nCouplerState AT %Q*:         UINT := 8;
	
	{attribute 'OPC.UA.DA':='0'}
	timer:			TON;
	
	{attribute 'OPC.UA.DA':='0'}
	trigger:		R_TRIG;	// To capture device INIT
	
	{attribute 'OPC.UA.DA':='0'}
	counter:		INT	:= 0; 	// Counter used to delay simulator initialisation
END_VAR

// Give simulator 20 cycles of idle until real device is ready.
IF counter < 20 THEN
	counter	:= counter + 1;
	RETURN;
END_IF

// Initialise the simulator, i.e. set pointers to the real device, etc.
IF NOT stat.bInitialised THEN
	// Set pointers to configuration and status
	ptrCfg	:= ADR(ptrDev^.cfg);
	ptrStat	:= ADR(ptrDev^.stat);

	// Check for NULL pointers in input parameters
	IF ptrCfg = 0  OR  ptrStat = 0 THEN
		stat.nErrorCode	:= E_SHUTTER_ERROR.SIM_NULL_POINTER;
		stat.sErrorText	:= 'ERROR: Input parameter is a NULL pointer';
		stat.sStatus	:= 'ERROR';
		RETURN;
	END_IF

	RPC_ResetConfig();	// Copy configuration from device
	
	timer(IN:=FALSE);
	timer(IN:=TRUE,PT:=UDINT_TO_TIME(100));	// Update almost immediately

	stat.nErrorCode	:= E_SHUTTER_ERROR.OK;
	stat.sErrorText	:= 'OK';
	stat.sStatus	:= 'OK';
	
	stat.bInitialised	:= TRUE;
	RETURN;
END_IF


// There are three triggers: 
// 	Detect device INIT or RESET
// 	RPC_ResetConfig() called (sets bUpdate to TRUE)
// 	Activation of switch

// Check for INIT or RESET trigger
trigger(CLK:=	(ptrStat^.sActionDesc = 'ActionInitExecute') OR 
				(ptrStat^.sActionDesc = 'ActionResetExecute'));

// Check if the control command has changed.
// If yes, set new outputs after a delay.
bSwitch := M_GetLogicalState(i_bSwitch, cfg.bActiveLowSwitch);

IF trigger.Q THEN
	RPC_ResetConfig();	// Copy configuration from device
ELSIF bSwitch <> bSwitchLast THEN
	// Switch value has changed. 
	bSwitchLast	:= bSwitch;	// Remember last switch value
	
	// Clear switches since the shutter is moving from one state to the other.
	bOpen	:= FALSE;
	bClosed	:= FALSE;

	// Update state after a delay.
	timer(IN:=FALSE);
	timer(IN:=TRUE,PT:=UDINT_TO_TIME(cfg.nDelay));
END_IF

// Execute the timer
timer();

// Set new outputs once the timer has expired
IF timer.Q THEN
	timer(IN:=FALSE);	// Reset timer
	SetState();
END_IF


(* Assign outputs *)
q_bFault		:= M_GetLogicalState(bFault, cfg.bActiveLowFault);
q_bOpen 		:= M_GetLogicalState(bOpen,	cfg.bActiveLowOpen);
q_bClosed 		:= M_GetLogicalState(bClosed,	cfg.bActiveLowClosed);
q_nCouplerState := nCouplerState;

METHOD M_GetLogicalState : BOOL
(*
	This method returns the state of the variable based on its 
	activeLow configuration.
	Syntax:
		bState	:= GetLogicalState (<var value>,  <activeLow cfg>);
		
	Example 1:
		var = TRUE;
		activeLow = FALSE;
		bState	:= GetLogicalState (TRUE,  FALSE); = TRUE

	Example 2:
		var = TRUE;
		activeLow = TRUE;
		bState	:= GetLogicalState (TRUE,  TRUE); = FALSE
*)
VAR_INPUT
	state:		BOOL;
	activeLow:	BOOL;
END_VAR
IF activeLow THEN
	M_GetLogicalState := NOT state;
ELSE
	M_GetLogicalState := state;
END_IF
END_METHOD

{attribute 'TcRpcEnable':='1'}
METHOD RPC_ResetConfig : INT
VAR_INPUT
END_VAR
cfg.bActiveLowOpen		:= ptrCfg^.bActiveLowOpen;
cfg.bActiveLowClosed	:= ptrCfg^.bActiveLowClosed;
cfg.bActiveLowFault		:= ptrCfg^.bActiveLowFault;
cfg.bActiveLowSwitch	:= ptrCfg^.bActiveLowSwitch;
cfg.nDelay				:= ptrCfg^.nTimeout / 2;	// Response delay = 1/2 of real shutter timeout
nCouplerState			:= 8;

// Reset Fault signal
bFault		:= FALSE;

// Set the Switch value to its initial state
bSwitch	:= ptrCfg^.bInitialState;

// Set Shutter state
SetState();

RPC_ResetConfig	:= E_SHUTTER_RPC_ERROR.OK;
END_METHOD

{attribute 'TcRpcEnable':='1'}
METHOD RPC_SetActiveLow_Closed : INT
VAR_INPUT
	bValue:	BOOL;
END_VAR
cfg.bActiveLowClosed:= bValue;

RPC_SetActiveLow_Closed	:= E_SHUTTER_RPC_ERROR.OK;
END_METHOD

{attribute 'TcRpcEnable':='1'}
METHOD RPC_SetActiveLow_Fault : INT
VAR_INPUT
	bValue:	BOOL;
END_VAR
cfg.bActiveLowFault	:= bValue;

RPC_SetActiveLow_Fault	:= E_SHUTTER_RPC_ERROR.OK;
END_METHOD

{attribute 'TcRpcEnable':='1'}
METHOD RPC_SetActiveLow_Open : INT
VAR_INPUT
	bValue:	BOOL;
END_VAR
cfg.bActiveLowOpen	:= bValue;

RPC_SetActiveLow_Open	:= E_SHUTTER_RPC_ERROR.OK;
END_METHOD

{attribute 'TcRpcEnable':='1'}
METHOD RPC_SetActiveLow_Switch : INT
VAR_INPUT
	bValue:	BOOL;
END_VAR
cfg.bActiveLowSwitch:= bValue;

RPC_SetActiveLow_Switch	:= E_SHUTTER_RPC_ERROR.OK;
END_METHOD

{attribute 'TcRpcEnable':='1'}
METHOD RPC_SetCouplerState : INT
VAR_INPUT
	nValue:	UINT;	// Coupler state, 8 = OPERATIONAL
END_VAR
nCouplerState	:= nValue;

RPC_SetCouplerState	:= E_SHUTTER_RPC_ERROR.OK;
END_METHOD

{attribute 'TcRpcEnable':='1'}
METHOD RPC_SetDelay : INT
VAR_INPUT
	nDelay:	UDINT;
END_VAR
cfg.nDelay	:= nDelay;

RPC_SetDelay	:= E_SHUTTER_RPC_ERROR.OK;
END_METHOD

{attribute 'TcRpcEnable':='1'}
METHOD RPC_SetFault : INT
VAR_INPUT
	bValue:	BOOL;
END_VAR
bFault:= M_GetLogicalState(bValue, cfg.bActiveLowFault);

RPC_SetFault	:= E_SHUTTER_RPC_ERROR.OK;
END_METHOD

METHOD SetState : BOOL
// Set Shutter state based on the input Switch value
VAR_INPUT
END_VAR
IF bSwitch THEN
	bOpen	:= TRUE;
	bClosed	:= FALSE;
ELSE
	bOpen	:= FALSE;
	bClosed	:= TRUE;
END_IF
END_METHOD

END_FUNCTION_BLOCK

// POUs/MAIN
PROGRAM MAIN
VAR
	// IMPORTANT:	In order to access RPC Calls via OPC UA, 
	//				attribute 'OPC.UA.DA':='1' is needed!!!
	{attribute 'OPC.UA.DA':='1'}
	Shutter001:		FB_SHUTTER;
	{attribute 'OPC.UA.DA':='1'}
	Shutter002:		FB_SHUTTER;
	{attribute 'OPC.UA.DA':='1'}
	Shutter003:		FB_SHUTTER;
	{attribute 'OPC.UA.DA':='1'}
	Shutter004:		FB_SHUTTER;
	{attribute 'OPC.UA.DA':='1'}
	Shutter005:		FB_SHUTTER;
	{attribute 'OPC.UA.DA':='1'}
	SIM_Shutter001:	FB_SIM_SHUTTER;
	{attribute 'OPC.UA.DA':='1'}
	SIM_Shutter002:	FB_SIM_SHUTTER;
	{attribute 'OPC.UA.DA':='1'}
	SIM_Shutter003:	FB_SIM_SHUTTER;
	{attribute 'OPC.UA.DA':='1'}
	SIM_Shutter004:	FB_SIM_SHUTTER;
	{attribute 'OPC.UA.DA':='1'}
	SIM_Shutter005:	FB_SIM_SHUTTER;
	
	ptrGUI_Shutters:	ARRAY [1..5] OF POINTER TO FB_SHUTTER	:= 
		[ADR(Shutter001), ADR(Shutter002), ADR(Shutter003), ADR(Shutter004), ADR(Shutter005)];
	nPtrIndex_Shutters:	INT	:= 1;

END_VAR

// Devices
Shutter001(in_sName:='Shutter001');
Shutter002(in_sName:='Shutter002', in_bActiveLowOpen:=TRUE, 	in_bActiveLowClosed:=TRUE);
Shutter003(in_sName:='Shutter003', in_bIgnoreClosed:=TRUE, 		in_bInitialState:=TRUE);
Shutter004(in_sName:='Shutter004', in_bActiveLowSwitch:=TRUE,	in_nTimeout:=500);
Shutter005(in_sName:='Shutter005', in_bActiveLowClosed:=TRUE);	// With PLC mappings this is a real shutter

// Simulators
SIM_Shutter001(ptrDev := ADR(Shutter001));
SIM_Shutter002(ptrDev := ADR(Shutter002));
SIM_Shutter003(ptrDev := ADR(Shutter003));
SIM_Shutter004(ptrDev := ADR(Shutter004));
SIM_Shutter005(ptrDev := ADR(Shutter005));	// With PLC mappings Shutter5 is linked to real HW.

END_PROGRAM

// VISUs/Templates/GUI_TEMPLATE_SHUTTER
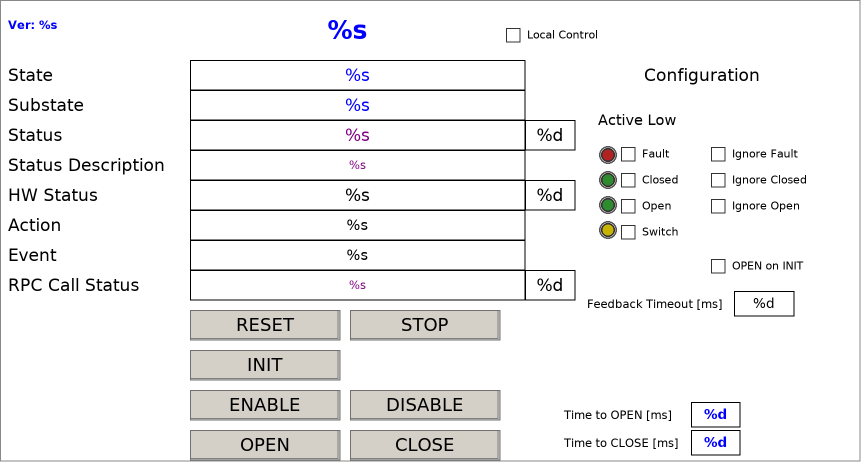
VISUALIZATION GUI_TEMPLATE_SHUTTER  // 861x462
VAR_IN_OUT
	m_Instance:	FB_SHUTTER;
END_VAR
    Rectangle (190,60 335x30), "%s", text variable: m_Instance.stat.sState
    Rectangle (190,90 335x30), "%s", text variable: m_Instance.stat.sSubstate
    Button (190,310 150x30), "RESET", input disabled if: (m_Instance.stat.bLocal = FALSE) <> 0
        OnMouseDown: execute { m_Instance.ctrl.nCommand :=E_SHUTTER_COMMAND.RESET; m_Instance.ctrl.bExecute := TRUE; }
    Button (190,350 150x30), "INIT", input disabled if: (m_Instance.stat.bLocal = FALSE) <> 0
        OnMouseDown: execute { m_Instance.ctrl.nCommand := E_SHUTTER_COMMAND.INIT; m_Instance.ctrl.bExecute := TRUE; }
    Button (350,310 150x30), "STOP", input disabled if: (m_Instance.stat.bLocal = FALSE) <> 0
        OnMouseDown: execute { m_Instance.ctrl.nCommand := E_SHUTTER_COMMAND.STOP; m_Instance.ctrl.bExecute := TRUE; }
    Button (190,390 150x30), "ENABLE", input disabled if: (m_Instance.stat.bLocal = FALSE) <> 0
        OnMouseDown: execute { m_Instance.ctrl.nCommand := E_SHUTTER_COMMAND.ENABLE; m_Instance.ctrl.bExecute := TRUE; }
    Button (350,390 150x30), "DISABLE", input disabled if: (m_Instance.stat.bLocal = FALSE) <> 0
        OnMouseDown: execute { m_Instance.ctrl.nCommand := E_SHUTTER_COMMAND.DISABLE; m_Instance.ctrl.bExecute := TRUE; }
    Button (190,430 150x30), "OPEN", input disabled if: (m_Instance.stat.bLocal = FALSE) <> 0
        OnMouseDown: execute { m_Instance.ctrl.nCommand := E_SHUTTER_COMMAND.OPEN; m_Instance.ctrl.bExecute := TRUE; }
    Button (350,430 150x30), "CLOSE", input disabled if: (m_Instance.stat.bLocal = FALSE) <> 0
        OnMouseDown: execute { m_Instance.ctrl.nCommand := E_SHUTTER_COMMAND.CLOSE; m_Instance.ctrl.bExecute := TRUE; }
    Rectangle (5,60 180x30), "State"
    Rectangle (5,90 180x30), "Substate"
    Rectangle (190,120 335x30), "%s", text variable: m_Instance.stat.sStatus
    Rectangle (190,150 335x30), "%s", text variable: m_Instance.stat.sErrorText
    Rectangle (5,120 180x30), "Status"
    Rectangle (5,150 180x30), "Status Description"
    Rectangle (190,210 335x30), "%s", text variable: m_Instance.stat.sActionDesc
    Rectangle (190,240 335x30), "%s", text variable: m_Instance.stat.sEventDesc
    Rectangle (190,180 335x30), "%s", text variable: m_Instance.stat.sHwStatus
    Rectangle (5,180 180x30), "HW Status"
    Rectangle (525,180 50x30), "%d", text variable: m_Instance.stat.nHwStatus
    Rectangle (5,210 180x30), "Action"
    Rectangle (5,240 180x30), "Event"
    Rectangle (190,12 315x35), "%s", text variable: m_Instance.cfg.sName
    Rectangle (525,120 50x30), "%d", text variable: m_Instance.stat.nStatus
    Checkbox (504,20 116x30), "Local Control", variable: m_Instance.stat.bLocal
    Rectangle (641,60 180x30), "Configuration"
    Rectangle (595,105 126x30), "Active Low"
    Checkbox (619,139 75x30), "Fault", variable: m_Instance.cfg.bActiveLowFault, input disabled if: (m_Instance.stat.bLocal = FALSE) <> 0
    Checkbox (709,139 110x30), "Ignore Fault", variable: m_Instance.cfg.bIgnoreFault, input disabled if: (m_Instance.stat.bLocal = FALSE) <> 0
    Checkbox (619,165 75x30), "Closed", variable: m_Instance.cfg.bActiveLowClosed, input disabled if: (m_Instance.stat.bLocal = FALSE) <> 0
    Checkbox (619,217 75x30), "Switch", variable: m_Instance.cfg.bActiveLowSwitch, input disabled if: (m_Instance.stat.bLocal = FALSE) <> 0
    Checkbox (709,251 150x30), "OPEN on INIT", tooltip "If selected, the default state of the shutter on INIT or DISABLE will be OPEN.", variable: m_Instance.cfg.bInitialState, input disabled if: (m_Instance.stat.bLocal = FALSE) <> 0
    Rectangle (734,291 60x25), "%d", tooltip "When controlling shutter, feedback signal should change within this period.", text variable: m_Instance.cfg.nTimeout, input disabled if: (m_Instance.stat.bLocal = FALSE) <> 0
        OnMouseDown: write the text variable via Default, min 0
    Rectangle (584,294 146x20), "Feedback Timeout [ms]"
    Checkbox (619,191 75x30), "Open", variable: m_Instance.cfg.bActiveLowOpen, input disabled if: (m_Instance.stat.bLocal = FALSE) <> 0
    Checkbox (709,165 110x30), "Ignore Closed", variable: m_Instance.cfg.bIgnoreClosed, input disabled if: (m_Instance.stat.bLocal = FALSE) <> 0
    Checkbox (709,191 110x30), "Ignore Open", variable: m_Instance.cfg.bIgnoreOpen, input disabled if: (m_Instance.stat.bLocal = FALSE) <> 0
    Rectangle (190,270 335x30), "%s", text variable: m_Instance.stat.sRPCErrorText
    Rectangle (5,270 180x30), "RPC Call Status"
    Rectangle (5,10 99x30), "Ver: %s", tooltip "'Shutter.library version'", text variable: m_Instance.stat.sLibVersion, input disabled if: true
    Rectangle (561,405 124x20), "Time to OPEN [ms]"
    Rectangle (561,433 124x20), "Time to CLOSE [ms]"
    Rectangle (691,402 49x25), "%d", tooltip "Last opening time [ms]. -1 means not open yet.", text variable: m_Instance.stat.nLastTimeToOpen
    Rectangle (691,430 49x25), "%d", tooltip "Last closing time [ms]. -1 means not closed yet.", text variable: m_Instance.stat.nLastTimeToClose
    Rectangle (525,270 50x30), "%d", tooltip "RPC Error Code 0 - OK", text variable: m_Instance.stat.nRpcErrorCode
    Lamp1 (598,145 20x20), tooltip "If ON, Fault signal is active.", variable: m_Instance.bFault, style: Lamp-Lamp1-Red
    Lamp1 (598,170 20x20), tooltip "If ON, Closed signal is active.", variable: m_Instance.bClosed, style: Lamp-Lamp1-Green
    Lamp1 (598,195 20x20), tooltip "If ON, Open signal is active.", variable: m_Instance.bOpen, style: Lamp-Lamp1-Green
    Lamp1 (598,220 20x20), tooltip "If ON, digital control output is high.", variable: m_Instance.q_bSwitch, style: Lamp-Lamp1-Yellow
END_VISUALIZATION

// VISUs/GUI_All
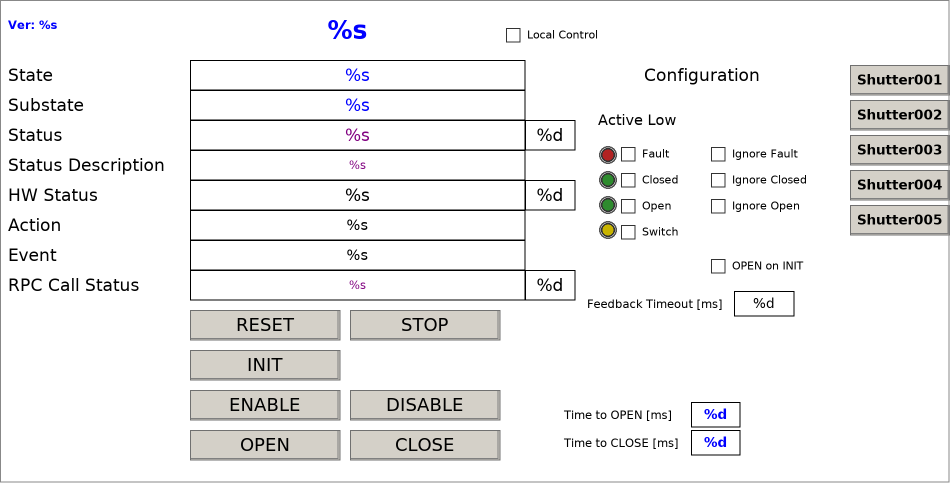
VISUALIZATION GUI_All  // 950x483
    Frame (0,0 827x483)
        shows GUI_TEMPLATE_SHUTTER(m_Instance := MAIN.ptrGUI_Shutters[MAIN.nPtrIndex_Shutters]^)
    Button (850,65 100x30), "Shutter001"
        OnMouseClick: execute { MAIN.nPtrIndex_Shutters:=1; }
    Button (850,100 100x30), "Shutter002"
        OnMouseClick: execute { MAIN.nPtrIndex_Shutters:=2; }
    Button (850,135 100x30), "Shutter003"
        OnMouseClick: execute { MAIN.nPtrIndex_Shutters:=3; }
    Button (850,170 100x30), "Shutter004"
        OnMouseClick: execute { MAIN.nPtrIndex_Shutters:=4; }
    Button (850,205 100x30), "Shutter005"
        OnMouseClick: execute { MAIN.nPtrIndex_Shutters:=5; }
END_VISUALIZATION

// VISUs/GUI_Shutter001
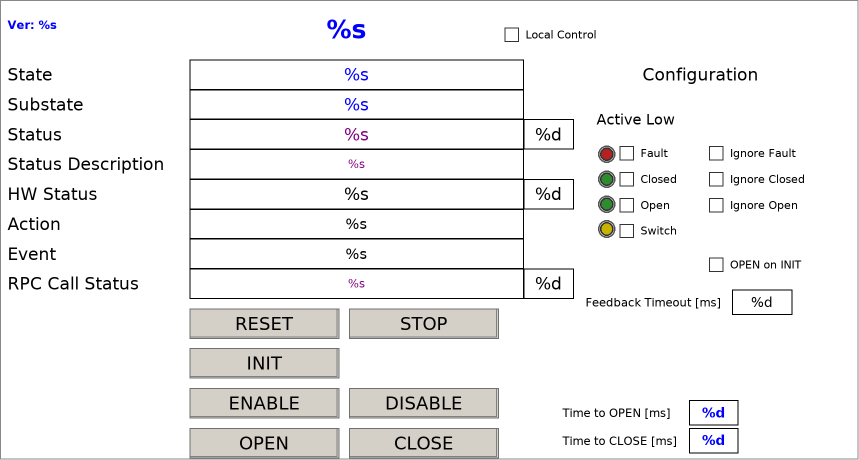
VISUALIZATION GUI_Shutter001  // 859x460
    Frame (0,0 859x460)
        shows GUI_TEMPLATE_SHUTTER(m_Instance := MAIN.Shutter001)
END_VISUALIZATION
